PROGRAM P_U01
VAR_INPUT
	auto_mode_on														: BOOL;

	shutdown_process													: BOOL;
	{attribute 'OPC.UA.DA' := '1'}  				                
	{attribute 'OPC.UA.DA.Access' := '1'}  				                
	co2_adsorption_interlock											: BOOL;
    /// <summary>PCV01</summary>
	{attribute 'OPC.UA.DA' := '1'}  				                
	vacuum_pres_control_valve											: REAL;
    /// <summary>PCV01</summary>                  	           
	{attribute 'OPC.UA.DA' := '1'}  				                
	vacuum_pres_control_valve_mode										: INT;			
    /// <summary>PCV02</summary>
	{attribute 'OPC.UA.DA' := '1'}  				                
	steam_flow_control_valve											: REAL;
    /// <summary>PCV02</summary>                  	           
	{attribute 'OPC.UA.DA' := '1'}  				                
	steam_flow_control_valve_mode										: INT;			
	{attribute 'OPC.UA.DA' := '1'}  				                
	{attribute 'OPC.UA.DA.Access' := '1'}  				                
	hot_sorbent_for_repressurization_interlock							: BOOL;
	{attribute 'OPC.UA.DA' := '1'}  				                
	{attribute 'OPC.UA.DA.Access' := '1'}  				                
	drainage_on															: BOOL;
	{attribute 'OPC.UA.DA' := '1'}  				                
	{attribute 'OPC.UA.DA.Access' := '1'}  				                
	repressurization_valve_with_steam_interlock							: BOOL;
	{attribute 'OPC.UA.DA' := '1'}  				                
	{attribute 'OPC.UA.DA.Access' := '1'}  				                
	door_open_with_steam_flow_interlock									: BOOL;
	{attribute 'OPC.UA.DA' := '1'}  				                
	{attribute 'OPC.UA.DA.Access' := '1'}  				                
	door_open_with_reactor_vacuum_interlock								: BOOL;
	{attribute 'OPC.UA.DA' := '1'}  				                
	{attribute 'OPC.UA.DA.Access' := '1'}  				                
	hot_reactor_condenser_interlock										: BOOL;
	{attribute 'OPC.UA.DA' := '1'}  				                
	{attribute 'OPC.UA.DA.Access' := '1'}  				                
	no_steam_unevacuated_reactor_interlock								: BOOL;
	{attribute 'OPC.UA.DA' := '1'}  				                
	{attribute 'OPC.UA.DA.Access' := '1'}  				                
	reactor_over_safe_pressure_limit_interlock							: BOOL;
	{attribute 'OPC.UA.DA' := '1'}  				                
	{attribute 'OPC.UA.DA.Access' := '1'}  				                
	reactor_over_safe_temperature_limit_interlock						: BOOL;
	
	/// <summary>XV10</summary>
	{attribute 'OPC.UA.DA' := '1'}  				                
	dead_air_inlet_valve												: BOOL;
	/// <summary>XV11</summary>
	{attribute 'OPC.UA.DA' := '1'}  				                
	product_line_ambient_valve											: BOOL;
    /// <summary>X01</summary>
	{attribute 'OPC.UA.DA' := '1'}  				                
	vacuum_liquid_loop_fan												: BOOL;
    /// <summary>P05</summary>
	{attribute 'OPC.UA.DA' := '1'}  				                
	vacuum_liquid_pump													: BOOL;
    /// <summary>P02</summary>
	{attribute 'OPC.UA.DA' := '1'}  				                
	vacuum_pump															: BOOL;
    /// <summary>XV04</summary>
	{attribute 'OPC.UA.DA' := '1'}  				                
	vacuum_pump_bypass_valve											: BOOL;
    /// <summary>XV03</summary>
	{attribute 'OPC.UA.DA' := '1'}  				                
	vacuum_pump_inlet_valve												: BOOL;
    /// <summary>P01</summary>
	{attribute 'OPC.UA.DA' := '1'}  				                
	steam_water_pump													: BOOL;
    /// <summary>B01</summary>
	{attribute 'OPC.UA.DA' := '1'}  				                
	boiler_package														: BOOL;
    /// <summary>P04</summary>
	{attribute 'OPC.UA.DA' := '1'}  				                
	condenser_pump														: BOOL;
    /// <summary>E01</summary>
	{attribute 'OPC.UA.DA' := '1'}  				                
	condenser_fan														: BOOL;
    /// <summary>P06</summary>
	{attribute 'OPC.UA.DA' := '1'}  				                
	vacuum_separator_drain_pump											: BOOL;
    /// <summary>PCV02</summary>
	steam_flow_control_valve_setpoint									: REAL;
	condenser_knockout_drain_adsorption_on									: BOOL;
	
END_VAR
VAR_OUTPUT
	utility_error														: STRING;
    /// <summary>XV10</summary>
	dead_air_inlet_valve_clear											: BOOL;
    /// <summary>XV11</summary>
	product_line_ambient_valve_clear									: BOOL;
    /// <summary>XV03</summary>
	vacuum_pump_inlet_valve_clear										: BOOL;
END_VAR
VAR

	fbWriteData															: FB_WritePersistentData;
	tonWriteData														: TON;
	bWriteData															: BOOL;
	
	sError																: STRING;
	sMessage															: STRING;
	sUtilityError														: STRING;
	sRS																	: STRING;
	iAxStep																: INT;
	i2Step																: INT;
	i3Step																: INT;
	i8Step																: INT;
	i9Step																: INT;
	iVfd_Speed															: INT;
	bCondition1															: BOOL;
	bCondition2															: BOOL;
	bCondition3															: BOOL;
	bAdsorptionActive													: BOOL;
	bComplete															: BOOL;
	bPreCheckDone														: BOOL;
	bTimer																: BOOL;
	bPass1																: BOOL;
	bPass2																: BOOL;
	bPass3																: BOOL;
	bAdsorptionTimer													: BOOL;
	bCloseXVValves														: BOOL;
	bRunSteamBypass														: BOOL;
	bVfd_Speed_Up														: BOOL;
	bCondenserKnockoutError												: BOOL;
	bVacuumSeparatorFillError											: BOOL;
	bVacuumSeparatorDrainError											: BOOL;
	rTime																: REAL;
	rSP																	: REAL;
	rPres																: REAL;
	tonTimer															: TON;
	tonAdsorptionTimer													: TON;
	tonBoilerCheck														: TON;
	tonVacuumInterlock													: TON;
	tonCondenserKODrain													: TON;
	tonVacuumSeparatorFill												: TON;
	tonVacuumSeparatorDrain												: TON;
	rtrigVacuumSeparator												: R_TRIG;
	rtrigKODrainValve													: R_TRIG;
	
	bCondenserFlowError													: BOOL;
	bCondensateFlowError												: BOOL;
	bFlowCalibrationDiffPresError										: BOOL;
	bInletLineTempError                                  	            : BOOL;
	bProductOutletCo2Error												: BOOL;
	bProductOutletFlowError												: BOOL;
	bProductOutletH2oError												: BOOL;
	bProductTempError                                   		       	: BOOL;
	bProductVacuumPresError												: BOOL;
	bProductVacuumTempError                              	          	: BOOL;
	bSteamFlowError														: BOOL;
	bSteamLinePresError													: BOOL;
	bSteamWaterTankLevelError											: BOOL;
	bVacuumPumpWaterFlowError											: BOOL;
	bVacuumPumpWaterTemp1Error											: BOOL;
	bVacuumSeparatorLevelError											: BOOL;
	bWaterFeedFlowError													: BOOL;
	bWaterScale1Error													: BOOL;
	bWaterScale2Error													: BOOL;
	bWaterScale3Error													: BOOL;

	fb_Vacuum_Pres_Control_Valve_PI										: FB_PI_Control();
	fb_Steam_Flow_Control_Valve_PI										: FB_PI_Control();
	
	fb_WaterScales_In													: FB_RateOfChange;
 	fb_WaterScales_Out													: FB_RateOfChange;
	{attribute 'OPC.UA.DA' := '1'} 
	water_scales_in_delta												: REAL;
	{attribute 'OPC.UA.DA' := '1'} 
	water_scales_out_delta												: REAL;
	{attribute 'OPC.UA.DA' := '1'} 
	water_scales_in_rate												: REAL;
	{attribute 'OPC.UA.DA' := '1'} 
	water_scales_out_rate												: REAL;
	{attribute 'OPC.UA.DA' := '1'} 
	water_scales_reset													: BOOL;
	fb_adsorp_product_wastewater										: FB_ChangeOfValue;
	
	{attribute 'OPC.UA.DA' := '1'}  				                
	pressure_drop_test													: BOOL;							// Pressure drop test flag

	{attribute 'OPC.UA.DA' := '1'}  				                
	interlock_condenser_steam_or										: BOOL;							// Override condenser pump & fan needing to be on when steam is flowing
	{attribute 'OPC.UA.DA' := '1'}  				                
	{attribute 'OPC.UA.DA.Access' := '1'}  				                
	interlock_condenser_steam_or_status									: BOOL;
	{attribute 'OPC.UA.DA' := '1'}  				                
	{attribute 'OPC.UA.DA.Access' := '1'}  				                
	condenser_steam_interlock											: BOOL;
	
	{attribute 'OPC.UA.DA' := '1'}  				                
	interlock_hot_reactor_condenser_or									: BOOL;							// Override dead air valve needing to be open if sorbent temp is high
	{attribute 'OPC.UA.DA' := '1'}  				                
	{attribute 'OPC.UA.DA.Access' := '1'}  				                
	interlock_hot_reactor_condenser_or_status							: BOOL;
	
	{attribute 'OPC.UA.DA' := '1'}  				                
	interlock_no_steam_unevacuated_reactor_or							: BOOL;							// Override no steam to unevacuated reactor
	{attribute 'OPC.UA.DA' := '1'}  				                
	{attribute 'OPC.UA.DA.Access' := '1'}  				                
	interlock_no_steam_unevacuated_reactor_or_status					: BOOL;
	
	{attribute 'OPC.UA.DA' := '1'}  				                
	interlock_cooling_with_vacuum_or									: BOOL;							// Override vacuum not running without cooling loop active
	{attribute 'OPC.UA.DA' := '1'}  				                
	{attribute 'OPC.UA.DA.Access' := '1'}  				                
	interlock_cooling_with_vacuum_or_status								: BOOL;
	{attribute 'OPC.UA.DA' := '1'}  				                
	{attribute 'OPC.UA.DA.Access' := '1'}  				                
	cooling_with_vacuum_interlock										: BOOL;
	
	{attribute 'OPC.UA.DA' := '1'}  				                
	interlock_separator_water_level_with_vacuum_or						: BOOL;							// Override vacuum not running while separator water level too high or too low
	{attribute 'OPC.UA.DA' := '1'}  				                
	{attribute 'OPC.UA.DA.Access' := '1'}  				                
	interlock_separator_water_level_with_vacuum_or_status				: BOOL;
	{attribute 'OPC.UA.DA' := '1'}  				                
	{attribute 'OPC.UA.DA.Access' := '1'}  				                
	separator_water_level_with_vacuum_interlock							: BOOL;
	
	{attribute 'OPC.UA.DA' := '1'}  				                
	interlock_cooling_loop_flow_with_vacuum_or							: BOOL;							// Override vacuum not running with insufficient cooling flow
	{attribute 'OPC.UA.DA' := '1'}  				                
	{attribute 'OPC.UA.DA.Access' := '1'}  				                
	interlock_cooling_loop_flow_with_vacuum_or_status					: BOOL;
	{attribute 'OPC.UA.DA' := '1'}  				                
	{attribute 'OPC.UA.DA.Access' := '1'}  				                
	cooling_loop_flow_with_vacuum_interlock								: BOOL;
	
	{attribute 'OPC.UA.DA' := '1'}  				                
	interlock_condensate_tank_level_for_steam_or						: BOOL;							// Override steam not running with condensate collection tank low 
	{attribute 'OPC.UA.DA' := '1'}  				                
	{attribute 'OPC.UA.DA.Access' := '1'}  				                
	interlock_condensate_tank_level_for_steam_or_status					: BOOL;
	{attribute 'OPC.UA.DA' := '1'}  				                
	{attribute 'OPC.UA.DA.Access' := '1'}  				                
	condensate_tank_level_for_steam_interlock							: BOOL;
	
	{attribute 'OPC.UA.DA' := '1'}  				                
	interlock_hot_sorbent_for_repressurization_or						: BOOL;							// Override repressurization not running if sorbent temp is high 
	{attribute 'OPC.UA.DA' := '1'}  				                
	{attribute 'OPC.UA.DA.Access' := '1'}  				                
	interlock_hot_sorbent_for_repressurization_or_status				: BOOL;
	
	{attribute 'OPC.UA.DA' := '1'}  				                
	interlock_reactor_over_safe_pressure_limit_or						: BOOL;							// Override reactor over safe pressure limit
	{attribute 'OPC.UA.DA' := '1'}  				                
	{attribute 'OPC.UA.DA.Access' := '1'}  				                
	interlock_reactor_over_safe_pressure_limit_or_status				: BOOL;
	
	{attribute 'OPC.UA.DA' := '1'}  				                
	interlock_reactor_over_safe_temperature_limit_or					: BOOL;							// Override reactor over safe temperature limit
	{attribute 'OPC.UA.DA' := '1'}  				                
	{attribute 'OPC.UA.DA.Access' := '1'}  				                
	interlock_reactor_over_safe_temperature_limit_or_status				: BOOL;
	
	{attribute 'OPC.UA.DA' := '1'}  				                
	interlock_repressurization_valve_with_steam_or						: BOOL;							// Override repressurization valve with steam flow
	{attribute 'OPC.UA.DA' := '1'}  				                
	{attribute 'OPC.UA.DA.Access' := '1'}  				                
	interlock_repressurization_valve_with_steam_or_status				: BOOL;
	
	{attribute 'OPC.UA.DA' := '1'}  				                
	interlock_door_open_with_steam_flow_or								: BOOL;							// Override door open with steam flow
	{attribute 'OPC.UA.DA' := '1'}  				                
	{attribute 'OPC.UA.DA.Access' := '1'}  				                
	interlock_door_open_with_steam_flow_or_status						: BOOL;
	
	{attribute 'OPC.UA.DA' := '1'}  				                
	interlock_door_open_with_reactor_vacuum_or							: BOOL;							// Override door open with reactor under vacuum
	{attribute 'OPC.UA.DA' := '1'}  				                
	{attribute 'OPC.UA.DA.Access' := '1'}  				                
	interlock_door_open_with_reactor_vacuum_or_status					: BOOL;
	
	{attribute 'OPC.UA.DA' := '1'}  				                
	interlock_co2_adsorption_or											: BOOL;							// Override co2 adsorption solenoids
	{attribute 'OPC.UA.DA' := '1'}  				                
	{attribute 'OPC.UA.DA.Access' := '1'}  				                
	interlock_co2_adsorption_or_status									: BOOL;
	
	{attribute 'OPC.UA.DA' := '1'}  				                
	interlock_condensate_pump_or										: BOOL;							// Override condensate pump
	{attribute 'OPC.UA.DA' := '1'}  				                
	{attribute 'OPC.UA.DA.Access' := '1'}  				                
	interlock_condensate_pump_or_status									: BOOL;
	{attribute 'OPC.UA.DA' := '1'}  				                
	{attribute 'OPC.UA.DA.Access' := '1'}  				                
	interlock_condensate_pump											: BOOL;
	
	{attribute 'OPC.UA.DA' := '1'}  				                
	vacuum_separator_drain_or_on										: BOOL;
	{attribute 'OPC.UA.DA' := '1'}  				                
	{attribute 'OPC.UA.DA.Access' := '1'}  				                
	vacuum_separator_drain_or_on_status									: BOOL;
	{attribute 'OPC.UA.DA' := '1'}  				                
	vacuum_separator_drain_or_off										: BOOL;
	{attribute 'OPC.UA.DA' := '1'}  				                
	{attribute 'OPC.UA.DA.Access' := '1'}  				                
	vacuum_separator_drain_or_off_status								: BOOL;

	{attribute 'OPC.UA.DA' := '1'}  				                
	reactor_drain_or_on													: BOOL;
	{attribute 'OPC.UA.DA' := '1'}  				                
	{attribute 'OPC.UA.DA.Access' := '1'}  				                
	reactor_drain_or_on_status											: BOOL;
	{attribute 'OPC.UA.DA' := '1'}  				                
	reactor_drain_or_off												: BOOL;
	{attribute 'OPC.UA.DA' := '1'}  				                
	{attribute 'OPC.UA.DA.Access' := '1'}  				                
	reactor_drain_or_off_status											: BOOL;

	{attribute 'OPC.UA.DA' := '1'}  				                
	condenser_knockout_drain_or_on										: BOOL;
	{attribute 'OPC.UA.DA' := '1'}  				                
	{attribute 'OPC.UA.DA.Access' := '1'}  				                
	condenser_knockout_drain_or_on_status								: BOOL;
	{attribute 'OPC.UA.DA' := '1'}  				                
	condenser_knockout_drain_or_off										: BOOL;
	{attribute 'OPC.UA.DA' := '1'}  				                
	{attribute 'OPC.UA.DA.Access' := '1'}  				                
	condenser_knockout_drain_or_off_status								: BOOL;

	{attribute 'OPC.UA.DA' := '1'}  				                
	{attribute 'OPC.UA.DA.Access' := '1'}  				                
	warmup_complete														: BOOL;
	{attribute 'OPC.UA.DA' := '1'}  				                
	{attribute 'OPC.UA.DA.Access' := '1'}  				                
	steam_bypass_complete												: BOOL;

	{attribute 'OPC.UA.DA' := '1'}  				                
	write_persistent_data												: BOOL;
	{attribute 'OPC.UA.DA' := '1'}  				                
	drainage_function_on_or												: BOOL;
	{attribute 'OPC.UA.DA' := '1'}  				                
	drainage_function_off_or											: BOOL;
	
	
	// PIDs
	steam_valve_pid 												: FB_CTRL_PID;
	steam_valve_pid_params											: ST_CTRL_PID_PARAMS;
	steam_valve_pid_mode											: E_CTRL_MODE := E_CTRL_MODE.eCTRL_MODE_MANUAL;
	steam_valve_pid_manual_sp										: LREAL := 50;   // Pressure SP value in manual mode
	steam_valve_pid_sp_value										: LREAL;  // Pressure SP value
	steam_valve_pid_actual_value									: LREAL;  // Presure Actual Value
	steam_valve_pid_out												: LREAL;  // valve control signal ( 0-100 %)
	steam_valve_pid_simulate_timer									: TON;
	steam_valve_pid_kp												: LREAL := 0.5;
	steam_valve_pid_tn												: TIME := T#5S;
	steam_valve_pid_tv												: TIME := T#0S;
	
	
	simulate_process												: FB_CTRL_PT2oscillation;
	simulate_process_params											: ST_CTRL_PT2oscillation_PARAMS ;
	simulate_process_kp												: REAL := 20;
	simulate_process_dumping_ration									: REAL := 0.5;
	simulate_process_tT0											: REAL := 0;
	
//	fb_MovingAverage												: FB_CTRL_MOVING_AVERAGE;
	moving_avg_in													: REAL;
	moving_avg_out													: LREAL;
	moving_avg_params												: ST_CTRL_MOVING_AVERAGE_PARAMS;
	moving_avg_array												: ARRAY[1..10] OF REAL;
	moving_avg_in_sim_timer											: TON;
	
	fbMovingAverage													: FB_MovingAverage;
	
	condenser_tank_capacity										: REAL;
	steam_delivery_tank_capacity										: REAL;
	condenser_tank_room_before_full										: REAL;
	steam_delivery_tank_before_empty										: REAL;
	
    /// <summary>LS01</summary>
	{attribute 'OPC.UA.DA' := '1'}  				                
	{attribute 'OPC.UA.DA.Access' := '1'}  				                
	product_condensate_drum_lsl									AT %I*	: BOOL;
    /// <summary>LS02</summary>
	{attribute 'OPC.UA.DA' := '1'}  				                
	{attribute 'OPC.UA.DA.Access' := '1'}  				                
	product_condensate_drum_lsh									AT %I*	: BOOL;

    /// <summary>B01</summary>
	{attribute 'OPC.UA.DA' := '1'}  				                
	{attribute 'OPC.UA.DA.Access' := '1'}  				                
	boiler_package_cmd_status											: BOOL;
    /// <summary>B01</summary>
	{attribute 'OPC.UA.DA' := '1'}  				                
	boiler_ready														: BOOL;
    /// <summary>boiler package</summary>
	B_01														AT %Q*	: BOOL;
    /// <summary>B01</summary>
	{attribute 'OPC.UA.DA' := '1'}  				                
	boiler_reset												AT %Q*	: BOOL;
	
    /// <summary>P02</summary>
	{attribute 'OPC.UA.DA' := '1'}  				                
	{attribute 'OPC.UA.DA.Access' := '1'}  				                
	steam_water_pump_cmd_status											: BOOL;
    /// <summary>vacuum pump</summary>
	P_01														AT %Q*	: BOOL;

    /// <summary>P02</summary>
	{attribute 'OPC.UA.DA' := '1'}  				                
	{attribute 'OPC.UA.DA.Access' := '1'}  				                
	vacuum_pump_cmd_status												: BOOL;
    /// <summary>vacuum pump</summary>
	P_02														AT %Q*	: BOOL;

    /// <summary>P03</summary>
	{attribute 'OPC.UA.DA' := '1'}  				                
	condensate_pump														: BOOL;
    /// <summary>P03</summary>
	{attribute 'OPC.UA.DA' := '1'}  				                
	{attribute 'OPC.UA.DA.Access' := '1'}  				                
	condensate_pump_cmd_status											: BOOL;
    /// <summary>condensate pump</summary>
	P_03														AT %Q*	: BOOL;

    /// <summary>P04</summary>
	{attribute 'OPC.UA.DA' := '1'}  				                
	{attribute 'OPC.UA.DA.Access' := '1'}  				                
	condenser_pump_cmd_status											: BOOL;
    /// <summary>condenser pump</summary>
	P_04														AT %Q*	: BOOL;

    /// <summary>P05</summary>
	{attribute 'OPC.UA.DA' := '1'}  				                
	{attribute 'OPC.UA.DA.Access' := '1'}  				                
	vacuum_liquid_pump_cmd_status										: BOOL;
    /// <summary>vacuum liquid pump</summary>
	P_05														AT %Q*	: BOOL;

    /// <summary>P06</summary>
	{attribute 'OPC.UA.DA' := '1'}  				                
	{attribute 'OPC.UA.DA.Access' := '1'}  				                
	vacuum_separator_drain_pump_cmd_status								: BOOL;
    /// <summary>vacuum cooling pump</summary>
	P_06														AT %Q*	: BOOL;

    /// <summary>E01</summary>
	{attribute 'OPC.UA.DA' := '1'}  				                
	{attribute 'OPC.UA.DA.Access' := '1'}  				                
	condenser_fan_cmd_status											: BOOL;
    /// <summary>condenser fan</summary>
	E_01														AT %Q*	: BOOL;

    /// <summary>X01</summary>
	{attribute 'OPC.UA.DA' := '1'}  				                
	{attribute 'OPC.UA.DA.Access' := '1'}  				                
	vacuum_liquid_loop_fan_cmd_status									: BOOL;
    /// <summary>vacuum liquid loop fan</summary>
	X_01														AT %Q*	: BOOL;

    /// <summary>AT02</summary>
	{attribute 'OPC.UA.DA' := '1'}  				                
	{attribute 'OPC.UA.DA.Access' := '1'}  				                
	product_outlet_co2													: REAL;
	{attribute 'OPC.UA.DA' := '1'}  				                
	{attribute 'OPC.UA.DA.Access' := '1'} 
    /// <summary>AT02</summary>
	product_outlet_co2_error											: BOOL;
    /// <summary>product outlet co2</summary>
	{attribute 'OPC.UA.DA' := '1'}  				                
	_ProductOutletCO2ErrorOff											: BOOL;
    /// <summary>AT02</summary>
	{attribute 'OPC.UA.DA' := '1'}  				                
	AT_02														AT %I*	: INT;
    /// <summary>AT02</summary>
	{attribute 'OPC.UA.DA' := '1'}  				                
	{attribute 'OPC.UA.DA.Access' := '1'}  				                
	AT_02_error													AT %I*	: BOOL;
    
	/// <summary>AT03</summary>
	{attribute 'OPC.UA.DA' := '1'}  				                
	{attribute 'OPC.UA.DA.Access' := '1'}  				                
	product_outlet_h2o													: REAL;
    /// <summary>AT03</summary>
	{attribute 'OPC.UA.DA' := '1'}  				                
	{attribute 'OPC.UA.DA.Access' := '1'}  				                
	product_outlet_h2o_error											: BOOL;
	/// <summary>AT03</summary>
	{attribute 'OPC.UA.DA' := '1'}  				                
	_ProductOutletH2OErrorOff											: BOOL;
    /// <summary>product outlet h2o</summary>
	AT_03														AT %I*	: INT;
    /// <summary>product outlet h2o</summary>
	{attribute 'OPC.UA.DA' := '1'}  				                
	{attribute 'OPC.UA.DA.Access' := '1'}  				                
	AT_03_error													AT %I*	: BOOL;

    /// <summary>FT02</summary>
	{attribute 'OPC.UA.DA' := '1'}  				                
	{attribute 'OPC.UA.DA.Access' := '1'}  					                
	product_outlet_flow													: REAL;
    /// <summary>FT02</summary>
	{attribute 'OPC.UA.DA' := '1'}  				                
	{attribute 'OPC.UA.DA.Access' := '1'}  				                
	product_outlet_flow_error											: BOOL;
    /// <summary>FT02</summary>
	{attribute 'OPC.UA.DA' := '1'}  				                
	_ProductOutletFlowErrorOff											: BOOL;
    /// <summary>product outlet flow</summary>
	FT_02														AT %I*	: INT;
    /// <summary>product outlet flow</summary>
	{attribute 'OPC.UA.DA' := '1'}  				                
	{attribute 'OPC.UA.DA.Access' := '1'}  				                
	FT_02_error													AT %I*	: BOOL;

    /// <summary>FT04</summary>
	{attribute 'OPC.UA.DA' := '1'}  				                
	{attribute 'OPC.UA.DA.Access' := '1'}  				                
	condensate_flow														: REAL;
    /// <summary>FT04</summary>
	{attribute 'OPC.UA.DA' := '1'}  				                
	{attribute 'OPC.UA.DA.Access' := '1'}  				                
	condensate_flow_error												: BOOL;
    /// <summary>FT04</summary>
	{attribute 'OPC.UA.DA' := '1'}  				                
	_CondensateFlowErrorOff												: BOOL;
    /// <summary>condensate flow</summary>
	FT_04														AT %I*	: INT;
    /// <summary>condensate flow</summary>
	{attribute 'OPC.UA.DA' := '1'}  				                
	{attribute 'OPC.UA.DA.Access' := '1'}  				                
	FT_04_error													AT %I*	: BOOL;

    /// <summary>FT05</summary>
	{attribute 'OPC.UA.DA' := '1'}  				                
	{attribute 'OPC.UA.DA.Access' := '1'}  					                
	tap_water_feed_flow													: REAL;
    /// <summary>FT05</summary>
	{attribute 'OPC.UA.DA' := '1'}  				                
	{attribute 'OPC.UA.DA.Access' := '1'}  				                
	tap_water_feed_flow_error											: BOOL;
    /// <summary>FT05</summary>
	{attribute 'OPC.UA.DA' := '1'}  				                
	_TapWaterFeedFlowErrorOff											: BOOL;
    /// <summary>tap water feed flow</summary>
	FT_05														AT %I*	: INT;
    /// <summary>tap water feed flow</summary>
	{attribute 'OPC.UA.DA' := '1'}  				                
	{attribute 'OPC.UA.DA.Access' := '1'}  				                
	FT_05_error													AT %I*	: BOOL;

    /// <summary>FT06</summary>
	{attribute 'OPC.UA.DA' := '1'}  				                
	{attribute 'OPC.UA.DA.Access' := '1'}  					                
	steam_flow															: REAL;
    /// <summary>FT06</summary>
	{attribute 'OPC.UA.DA' := '1'}  				                
	{attribute 'OPC.UA.DA.Access' := '1'}  				                
	steam_flow_error													: BOOL;
    /// <summary>FT06</summary>
	{attribute 'OPC.UA.DA' := '1'}  				                
	_SteamFlowErrorOff													: BOOL;
    /// <summary>steam flow</summary>
	FT_06														AT %I*	: INT;
    /// <summary>steam flow</summary>
	{attribute 'OPC.UA.DA' := '1'}  				                
	{attribute 'OPC.UA.DA.Access' := '1'}  				                
	FT_06_error													AT %I*	: BOOL;

    /// <summary>FT07</summary>
	{attribute 'OPC.UA.DA' := '1'}  				                
	{attribute 'OPC.UA.DA.Access' := '1'}  					                
	vacuum_pump_water_flow												: REAL;
    /// <summary>FT07</summary>
	{attribute 'OPC.UA.DA' := '1'}  				                
	{attribute 'OPC.UA.DA.Access' := '1'}  				                
	vacuum_pump_water_flow_error										: BOOL;
    /// <summary>FT07</summary>
	{attribute 'OPC.UA.DA' := '1'}  				                
	_VacuumPumpWaterFlowErrorOff										: BOOL;
    /// <summary>vacuum pump water flow</summary>
	FT_07														AT %I*	: INT;
    /// <summary>vacuum pump water flow</summary>
    /// <summary>FT07</summary>
	{attribute 'OPC.UA.DA' := '1'}  				                
	{attribute 'OPC.UA.DA.Access' := '1'}  				                
	FT_07_error													AT %I*	: BOOL;

    /// <summary>FT08</summary>
	{attribute 'OPC.UA.DA' := '1'}  				                
	{attribute 'OPC.UA.DA.Access' := '1'}  					                
	condenser_flow														: REAL;
    /// <summary>FT08</summary>
	{attribute 'OPC.UA.DA' := '1'}  				                
	{attribute 'OPC.UA.DA.Access' := '1'}  				                
	condenser_flow_error												: BOOL;
    /// <summary>FT08</summary>
	{attribute 'OPC.UA.DA' := '1'}  				                
	_CondenserFlowErrorOff												: BOOL;
    /// <summary>vacuum pump water flow</summary>
	FT_08														AT %I*	: INT;
    /// <summary>vacuum pump water flow</summary>
    /// <summary>FT08</summary>
	{attribute 'OPC.UA.DA' := '1'}  				                
	{attribute 'OPC.UA.DA.Access' := '1'}  				                
	FT_08_error													AT %I*	: BOOL;

    /// <summary>LT01</summary>
	{attribute 'OPC.UA.DA' := '1'}  				                
	{attribute 'OPC.UA.DA.Access' := '1'}  					                
	steam_water_tank_level												: REAL;
    /// <summary>LT01</summary>
	{attribute 'OPC.UA.DA' := '1'}  				                
	{attribute 'OPC.UA.DA.Access' := '1'}  				                
	steam_water_tank_level_error										: BOOL;
    /// <summary>LT01</summary>
	{attribute 'OPC.UA.DA' := '1'}  				                
	_SteamWaterTankLevelErrorOff										: BOOL;
    /// <summary>steam water tank level</summary>
	LT_01														AT %I*	: INT;
    /// <summary>steam water tank level</summary>
    /// <summary>LT01</summary>
	{attribute 'OPC.UA.DA' := '1'}  				                
	{attribute 'OPC.UA.DA.Access' := '1'}  				                
	LT_01_error													AT %I*	: BOOL;

    /// <summary>LT02</summary>
	{attribute 'OPC.UA.DA' := '1'}  				                
	{attribute 'OPC.UA.DA.Access' := '1'}  					                
	vacuum_separator_level												: REAL;
    /// <summary>LT02</summary>
	{attribute 'OPC.UA.DA' := '1'}  				                
	{attribute 'OPC.UA.DA.Access' := '1'}  				                
	vacuum_separator_level_error										: BOOL;
    /// <summary>LT02</summary>
	{attribute 'OPC.UA.DA' := '1'}  				                
	_VacuumSeparatorLevelErrorOff										: BOOL;
    /// <summary>vacuum separator level</summary>
	LT_02														AT %I*	: INT;
    /// <summary>vacuum separator level</summary>
    /// <summary>LT02</summary>
	{attribute 'OPC.UA.DA' := '1'}  				                
	{attribute 'OPC.UA.DA.Access' := '1'}  				                
	LT_02_error													AT %I*	: BOOL;

    /// <summary>PT04</summary>
	{attribute 'OPC.UA.DA' := '1'}  				                
	{attribute 'OPC.UA.DA.Access' := '1'}  				                
	product_vacuum_pres													: REAL;
    /// <summary>PT04</summary>
	{attribute 'OPC.UA.DA' := '1'}  				                
	{attribute 'OPC.UA.DA.Access' := '1'}  				                
	product_vacuum_pres_error											: BOOL;
    /// <summary>PT04</summary>
	{attribute 'OPC.UA.DA' := '1'}  				                
	_ProductVacuumPresErrorOff											: BOOL;
    /// <summary>product vacuum pres</summary>
	PT_04														AT %I*	: INT;
    /// <summary>product vacuum pres</summary>
    /// <summary>PT04</summary>
	{attribute 'OPC.UA.DA' := '1'}  				                
	{attribute 'OPC.UA.DA.Access' := '1'}  				                
	PT_04_error													AT %I*	: BOOL;

    /// <summary>PT07</summary>
	{attribute 'OPC.UA.DA' := '1'}  				                
	{attribute 'OPC.UA.DA.Access' := '1'}  				                
	steam_line_pres														: REAL;
    /// <summary>PT07</summary>
	{attribute 'OPC.UA.DA' := '1'}  				                
	{attribute 'OPC.UA.DA.Access' := '1'}  				                
	steam_line_pres_error												: BOOL;
    /// <summary>PT07</summary>
	{attribute 'OPC.UA.DA' := '1'}  				                
	_SteamLinePresErrorOff												: BOOL;
    /// <summary>steam line pres</summary>
	PT_07														AT %I*	: INT;
    /// <summary>steam line pres</summary>
	{attribute 'OPC.UA.DA' := '1'}  				                
	{attribute 'OPC.UA.DA.Access' := '1'}  				                
	PT_07_error													AT %I*	: BOOL;

    /// <summary>PDT04</summary>
	{attribute 'OPC.UA.DA' := '1'}  				                
	{attribute 'OPC.UA.DA.Access' := '1'}  				                
	flow_calibration_diff_pres											: REAL;
    /// <summary>PDT04</summary>
	{attribute 'OPC.UA.DA' := '1'}  				                
	{attribute 'OPC.UA.DA.Access' := '1'}  				                
	flow_calibration_diff_pres_error									: BOOL;
    /// <summary>PDT04</summary>
	{attribute 'OPC.UA.DA' := '1'}  				                
	_FlowCalibrationDiffPresErrorOff									: BOOL;
    /// <summary>flow calibration diff pres</summary>
	PDT_04														AT %I*	: INT;
    /// <summary>flow calibration diff pres</summary>
	{attribute 'OPC.UA.DA' := '1'}  				                
	{attribute 'OPC.UA.DA.Access' := '1'}  				                
	PDT_04_error												AT %I*	: BOOL;

    /// <summary>TT02</summary>
	{attribute 'OPC.UA.DA' := '1'}  				                
	{attribute 'OPC.UA.DA.Access' := '1'}  				                
	product_temp														: REAL;
    /// <summary>TT02</summary>
	{attribute 'OPC.UA.DA' := '1'}  				                
	{attribute 'OPC.UA.DA.Access' := '1'}  				                
	product_temp_error													: BOOL;
	{attribute 'OPC.UA.DA' := '1'}  				                
	_ProductTempErrorOff												: BOOL;
    /// <summary>product temp</summary>
	TT_02														AT %I*	: INT;
    /// <summary>product temp</summary>
	{attribute 'OPC.UA.DA' := '1'}  				                
	{attribute 'OPC.UA.DA.Access' := '1'}  				                
	TT_02_error													AT %I*	: BOOL;

    /// <summary>TT03</summary>
	{attribute 'OPC.UA.DA' := '1'}  				                
	{attribute 'OPC.UA.DA.Access' := '1'}  				                
	product_vacuum_temp													: REAL;
    /// <summary>TT03</summary>
	{attribute 'OPC.UA.DA' := '1'}  				                
	{attribute 'OPC.UA.DA.Access' := '1'}  				                
	product_vacuum_temp_error											: BOOL;
    /// <summary>TT03</summary>
	{attribute 'OPC.UA.DA' := '1'}  				                
	_ProductVacuumTempOff												: BOOL;
    /// <summary>product vacuum temp</summary>
	TT_03														AT %I*	: INT;
    /// <summary>product vacuum temp</summary>
	{attribute 'OPC.UA.DA' := '1'}  				                
	{attribute 'OPC.UA.DA.Access' := '1'}  				                
	TT_03_error													AT %I*	: BOOL;

    /// <summary>TT06</summary>
	{attribute 'OPC.UA.DA' := '1'}  				                
	{attribute 'OPC.UA.DA.Access' := '1'}  				                
	inlet_line_temp														: REAL;
    /// <summary>TT06</summary>
	{attribute 'OPC.UA.DA' := '1'}  				                
	{attribute 'OPC.UA.DA.Access' := '1'}  				                
	inlet_line_temp_error												: BOOL;
    /// <summary>TT06</summary>
	{attribute 'OPC.UA.DA' := '1'}  				                
	_InletLineTempErrorOff												: BOOL;
    /// <summary>inlet line temp</summary>
	TT_06														AT %I*	: INT;
    /// <summary>inlet line temp</summary>
	{attribute 'OPC.UA.DA' := '1'}  				                
	{attribute 'OPC.UA.DA.Access' := '1'}  				                
	TT_06_error													AT %I*	: BOOL;

    /// <summary>TT10</summary>
	{attribute 'OPC.UA.DA' := '1'}  				                
	{attribute 'OPC.UA.DA.Access' := '1'}  				                
	vacuum_pump_water_temp_1											: REAL;
    /// <summary>TT10</summary>
	{attribute 'OPC.UA.DA' := '1'}  				                
	{attribute 'OPC.UA.DA.Access' := '1'}  				                
	vacuum_pump_water_temp_1_error										: BOOL;
    /// <summary>TT10</summary>
	{attribute 'OPC.UA.DA' := '1'}  				                
	_VacuumPumpWaterTemp1ErrorOff										: BOOL;
    /// <summary>vacuum pump water temp 1</summary>
	TT_10														AT %I*	: INT;
    /// <summary>vacuum pump water temp 1</summary>
	{attribute 'OPC.UA.DA' := '1'}  				                
	{attribute 'OPC.UA.DA.Access' := '1'}  				                
	TT_10_error													AT %I*	: BOOL;
	
    /// <summary>TT11</summary>
	{attribute 'OPC.UA.DA' := '1'}  				                
	{attribute 'OPC.UA.DA.Access' := '1'}  				                
	vacuum_pump_water_temp_2											: REAL;
    /// <summary>TT11</summary>
	{attribute 'OPC.UA.DA' := '1'}  				                
	{attribute 'OPC.UA.DA.Access' := '1'}  				                
	vacuum_pump_water_temp_2_error										: BOOL;
    /// <summary>TT11</summary>
	{attribute 'OPC.UA.DA' := '1'}  				                
	_VacuumPumpWaterTemp2ErrorOff										: BOOL;
    /// <summary>vacuum pump water temp 2</summary>
	TT_11														AT %I*	: INT;
    /// <summary>vacuum pump water temp 2</summary>
	{attribute 'OPC.UA.DA' := '1'}  				                
	{attribute 'OPC.UA.DA.Access' := '1'}  				                
	TT_11_error													AT %I*	: BOOL;

    /// <summary>XV03</summary>
	{attribute 'OPC.UA.DA' := '1'}  				                
	{attribute 'OPC.UA.DA.Access' := '1'}  				                
	vacuum_pump_inlet_valve_open_cmd_status								: BOOL;
    /// <summary>XV03</summary>
	{attribute 'OPC.UA.DA' := '1'}  				                
	{attribute 'OPC.UA.DA.Access' := '1'}  				                
	vacuum_pump_inlet_valve_open								AT %I*	: BOOL;
    /// <summary>XV03</summary>
	{attribute 'OPC.UA.DA' := '1'}  				                
	{attribute 'OPC.UA.DA.Access' := '1'}  				                
	vacuum_pump_inlet_valve_closed								AT %I*	: BOOL;
    /// <summary>vacuum pump inlet valve</summary>
	XV_03														AT %Q*	: BOOL;
	
    /// <summary>XV04</summary>
	{attribute 'OPC.UA.DA' := '1'}  				                
	{attribute 'OPC.UA.DA.Access' := '1'}  				                
	vacuum_pump_bypass_valve_open_cmd_status							: BOOL;
    /// <summary>XV04</summary>
	{attribute 'OPC.UA.DA' := '1'}  				                
	{attribute 'OPC.UA.DA.Access' := '1'}  				                
	vacuum_pump_bypass_valve_open								AT %I*	: BOOL;
    /// <summary>XV04</summary>
	{attribute 'OPC.UA.DA' := '1'}  				                
	{attribute 'OPC.UA.DA.Access' := '1'}  				                
	vacuum_pump_bypass_valve_closed								AT %I*	: BOOL;
    /// <summary>vacuum pump bypass valve</summary>
	XV_04														AT %Q*	: BOOL;
    /// <summary>XV04</summary>
	vacuum_pump_bypass_valve_clear										: BOOL;
	
    /// <summary>XV06</summary>
	{attribute 'OPC.UA.DA' := '1'}  				                
	knockout_drain_valve												: BOOL;
    /// <summary>XV06</summary>
	{attribute 'OPC.UA.DA' := '1'}  				                
	{attribute 'OPC.UA.DA.Access' := '1'}  				                
	knockout_drain_valve_open_cmd_status								: BOOL;
    /// <summary>XV06</summary>
	{attribute 'OPC.UA.DA' := '1'}  				                
	{attribute 'OPC.UA.DA.Access' := '1'}  				                
	knockout_drain_valve_open									AT %I*	: BOOL;
    /// <summary>XV06</summary>
	{attribute 'OPC.UA.DA' := '1'}  				                
	{attribute 'OPC.UA.DA.Access' := '1'}  				                
	knockout_drain_valve_closed									AT %I*	: BOOL;
    /// <summary>knockout drain valve</summary>
	XV_06														AT %Q*	: BOOL;
    /// <summary>XV06</summary>
	knockout_drain_valve_clear											: BOOL;
	
    /// <summary>XV10</summary>
	{attribute 'OPC.UA.DA' := '1'}  				                
	{attribute 'OPC.UA.DA.Access' := '1'}  				                
	dead_air_inlet_valve_open_cmd_status								: BOOL;
    /// <summary>XV10</summary>
	{attribute 'OPC.UA.DA' := '1'}  				                
	{attribute 'OPC.UA.DA.Access' := '1'}  				                
	dead_air_inlet_valve_open									AT %I*	: BOOL;
    /// <summary>XV10</summary>
	{attribute 'OPC.UA.DA' := '1'}  				                
	{attribute 'OPC.UA.DA.Access' := '1'}  				                
	dead_air_inlet_valve_closed 								AT %I*	: BOOL;
    /// <summary>dead air inlet valve</summary>
	XV_10														AT %Q*	: BOOL;

    /// <summary>XV11</summary>
	{attribute 'OPC.UA.DA' := '1'}  				                
	{attribute 'OPC.UA.DA.Access' := '1'}  				                
	product_line_ambient_valve_cmd_status								: BOOL;
    /// <summary>XV11</summary>
	{attribute 'OPC.UA.DA' := '1'}  				                
	{attribute 'OPC.UA.DA.Access' := '1'}  				                
	product_line_ambient_valve_product 							AT %I*	: BOOL;				///@@@ Assuming open valve is Product
    /// <summary>XV11</summary>
	{attribute 'OPC.UA.DA' := '1'}  				                
	{attribute 'OPC.UA.DA.Access' := '1'}  				                
	product_line_ambient_valve_ambient							AT %I*	: BOOL;				///@@@ Assuming closed valve is Ambient
    /// <summary>product line ambient valve</summary>
	XV_11														AT %Q*	: BOOL;

	/// <summary>XV12</summary>
	{attribute 'OPC.UA.DA' := '1'}  				                
	tap_water_feed_valve												: BOOL;
    /// <summary>XV11</summary>
	{attribute 'OPC.UA.DA' := '1'}  				                
	{attribute 'OPC.UA.DA.Access' := '1'}  				                
	tap_water_feed_valve_cmd_status										: BOOL;
	XV_12														AT %Q*	: BOOL;

	/// <summary>XV13</summary>
	{attribute 'OPC.UA.DA' := '1'}  				                
	separator_drain_valve												: BOOL;
    /// <summary>XV13</summary>
	{attribute 'OPC.UA.DA' := '1'}  				                
	{attribute 'OPC.UA.DA.Access' := '1'}  				                
	separator_drain_valve_open_cmd_status								: BOOL;
    /// <summary>XV13</summary>
	{attribute 'OPC.UA.DA' := '1'}  				                
	{attribute 'OPC.UA.DA.Access' := '1'}  				                
	separator_drain_valve_open									AT %I*	: BOOL;
    /// <summary>XV13</summary>
	{attribute 'OPC.UA.DA' := '1'}  				                
	{attribute 'OPC.UA.DA.Access' := '1'}  				                
	separator_drain_valve_closed 								AT %I*	: BOOL;
    /// <summary>dead air inlet valve</summary>
	XV_13														AT %Q*	: BOOL;
    /// <summary>XV13</summary>
	separator_drain_valve_clear											: BOOL;

	/// <summary>XV14</summary>
	{attribute 'OPC.UA.DA' := '1'}  				                
	steam_water_reservoir_valve											: BOOL;
    /// <summary>XV14</summary>
	{attribute 'OPC.UA.DA' := '1'}  				                
	{attribute 'OPC.UA.DA.Access' := '1'}  				                
	steam_water_reservoir_valve_cmd_status								: BOOL;
    /// <summary>steam water reservoir valve</summary>
	XV_14														AT %Q*	: BOOL;

    /// <summary>PCV01</summary>
	vacuum_pres_control_valve_open										: BOOL;
    /// <summary>PCV01</summary>
	vacuum_pres_control_valve_closed									: BOOL;
    /// <summary>PCV01</summary>
	{attribute 'OPC.UA.DA' := '1'}  				                
	{attribute 'OPC.UA.DA.Access' := '1'}  				                
	vacuum_pres_control_valve_position									: REAL;
    /// <summary>PCV01</summary>
	{attribute 'OPC.UA.DA' := '1'}  				                
	{attribute 'OPC.UA.DA.Access' := '1'}  				                
	vacuum_pres_control_valve_position_error					AT %I*	: BOOL;
    /// <summary>vacuum pressure control valve</summary>
	PCV_01														AT %Q*	: INT;
    /// <summary>vacuum pressure control valve</summary>
	{attribute 'OPC.UA.DA' := '1'}  				                
	{attribute 'OPC.UA.DA.Access' := '1'}  				                
	PCV_01_position												AT %I*	: INT;
    /// <summary>PCV01</summary>                  	           
	{attribute 'OPC.UA.DA' := '1'}  				                
	{attribute 'OPC.UA.DA.Access' := '1'}  				                
	vacuum_pres_control_valve_current_mode								: INT;			
    /// <summary>PCV01</summary>                  	           
	vacuum_pres_control_valve_kp										: REAL		:= 0.01; 
    /// <summary>PCV01</summary>                  	           
	vacuum_pres_control_valve_ki										: REAL		:= 0.01;
    /// <summary>PCV01</summary>                  	           
	vacuum_pres_control_valve_loop_time									: REAL		:= 2000;
    /// <summary>PCV01</summary>                  	           
	vacuum_pres_control_valve_iband										: REAL		:= 6;
    /// <summary>PCV01</summary>                  	           
	vacuum_pres_control_valve_base										: INT		:= 13110;
    /// <summary>PCV01</summary>                  	           
	vacuum_pres_control_valve_base_adjust								: INT		:= 10;
	
    /// <summary>PCV02</summary>
	steam_flow_control_valve_open										: BOOL;
    /// <summary>PCV02</summary>
	steam_flow_control_valve_closed										: BOOL;
    /// <summary>PCV02</summary>
	{attribute 'OPC.UA.DA' := '1'}  				                
	{attribute 'OPC.UA.DA.Access' := '1'}  				                
	steam_flow_control_valve_position									: REAL;
    /// <summary>PCV02</summary>
	{attribute 'OPC.UA.DA' := '1'}  				                
	{attribute 'OPC.UA.DA.Access' := '1'}  				                
	steam_flow_control_valve_position_error								: BOOL;
    /// <summary>steam flow control valve</summary>
	PCV_02														AT %Q*	: INT;
    /// <summary>steam flow control valve</summary>
	{attribute 'OPC.UA.DA' := '1'}  				                
	{attribute 'OPC.UA.DA.Access' := '1'}  				                
	PCV_02_position												AT %I*	: INT;
    /// <summary>PCV02</summary>                  	           
	{attribute 'OPC.UA.DA' := '1'}  				                
	{attribute 'OPC.UA.DA.Access' := '1'}  				                
	steam_flow_control_valve_current_mode								: INT;			
    /// <summary>PCV02</summary>                  	           
	steam_flow_control_valve_kp											: REAL		:= 0.01; 
    /// <summary>PCV02</summary>                  	           
	steam_flow_control_valve_ki											: REAL		:= 0.01;
    /// <summary>PCV02</summary>                  	           
	steam_flow_control_valve_loop_time									: REAL		:= 2000;
    /// <summary>PCV02</summary>                  	           
	steam_flow_control_valve_iband										: REAL		:= 6;
    /// <summary>PCV02</summary>                  	           
	steam_flow_control_valve_base										: INT		:= 13110;
    /// <summary>PCV02</summary>                  	           
	steam_flow_control_valve_base_adjust								: INT		:= 10;
	
	{attribute 'OPC.UA.DA' := '1'}  				                
	{attribute 'OPC.UA.DA.Access' := '1'}  				                
	l1_current_240														: REAL;
	{attribute 'OPC.UA.DA' := '1'}  				                
	{attribute 'OPC.UA.DA.Access' := '1'}  				                
	l1_current_240_error										AT %I*	: BOOL;
	IT1															AT %I*	: INT;
	{attribute 'OPC.UA.DA' := '1'}  				                
	{attribute 'OPC.UA.DA.Access' := '1'}  				                
	l2_current_240														: REAL;
	{attribute 'OPC.UA.DA' := '1'}  				                
	{attribute 'OPC.UA.DA.Access' := '1'}  				                
	l2_current_240_error										AT %I*	: BOOL;
	IT2															AT %I*	: INT;
	{attribute 'OPC.UA.DA' := '1'}  				                
	{attribute 'OPC.UA.DA.Access' := '1'}  				                
	l3_current_240														: REAL;
	{attribute 'OPC.UA.DA' := '1'}  				                
	{attribute 'OPC.UA.DA.Access' := '1'}  				                
	l3_current_240_error										AT %I*	: BOOL;
	IT3															AT %I*	: INT;
	
	{attribute 'OPC.UA.DA' := '1'}  				                
	{attribute 'OPC.UA.DA.Access' := '1'}  				                
	l1_voltage_240														: REAL;
	{attribute 'OPC.UA.DA' := '1'}  				                
	{attribute 'OPC.UA.DA.Access' := '1'}  				                
	l1_voltage_240_error										AT %I*	: BOOL;
	{attribute 'OPC.UA.DA' := '1'}  				                
	VT1															AT %I*	: INT;
	{attribute 'OPC.UA.DA' := '1'}  				                
	l2_voltage_240														: REAL;
	{attribute 'OPC.UA.DA' := '1'}  				                
	{attribute 'OPC.UA.DA.Access' := '1'}  				                
	l2_voltage_240_error										AT %I*	: BOOL;
	{attribute 'OPC.UA.DA' := '1'}  				                
	VT2															AT %I*	: INT;
	{attribute 'OPC.UA.DA' := '1'}  				                
	l3_voltage_240														: REAL;
	{attribute 'OPC.UA.DA' := '1'}  				                
	{attribute 'OPC.UA.DA.Access' := '1'}  				                
	l3_voltage_240_error										AT %I*	: BOOL;
	{attribute 'OPC.UA.DA' := '1'}  				                
	VT3															AT %I*	: INT;
	
	{attribute 'OPC.UA.DA' := '1'}  				                
	{attribute 'OPC.UA.DA.Access' := '1'}  				                
	l1_current_120														: REAL;
	{attribute 'OPC.UA.DA' := '1'}  				                
	{attribute 'OPC.UA.DA.Access' := '1'}  				                
	l1_current_120_error										AT %I*	: BOOL;
	IT4															AT %I*	: INT;
	
	{attribute 'OPC.UA.DA' := '1'}  				                
	{attribute 'OPC.UA.DA.Access' := '1'}  				                
	l1_voltage_120														: REAL;
	{attribute 'OPC.UA.DA' := '1'}  				                
	{attribute 'OPC.UA.DA.Access' := '1'}  				                
	l1_voltage_120_error										AT %I*	: BOOL;
	VT4															AT %I*	: INT;
	
	{attribute 'OPC.UA.DA' := '1'}  				                
	{attribute 'OPC.UA.DA.Access' := '1'}  				                
	l1_current_boiler													: REAL;
	{attribute 'OPC.UA.DA' := '1'}  				                
	{attribute 'OPC.UA.DA.Access' := '1'}  				                
	l1_current_boiler_error										AT %I*	: BOOL;
	IT_boiler_01												AT %I*	: INT;
	{attribute 'OPC.UA.DA' := '1'}  				                
	{attribute 'OPC.UA.DA.Access' := '1'}  				                
	l2_current_boiler													: REAL;
	{attribute 'OPC.UA.DA' := '1'}  				                
	{attribute 'OPC.UA.DA.Access' := '1'}  				                
	l2_current_boiler_error										AT %I*	: BOOL;
	IT_boiler_02												AT %I*	: INT;
	{attribute 'OPC.UA.DA' := '1'}  				                
	{attribute 'OPC.UA.DA.Access' := '1'}  				                
	l3_current_boiler													: REAL;
	{attribute 'OPC.UA.DA' := '1'}  				                
	{attribute 'OPC.UA.DA.Access' := '1'}  				                
	l3_current_boiler_error										AT %I*	: BOOL;
	IT_boiler_03												AT %I*	: INT;
	
	//== Water Scales ====
	  /// <summary>WI01</summary>
	{attribute 'OPC.UA.DA' := '1'}  				                
	{attribute 'OPC.UA.DA.Access' := '1'}  				                
	water_scale_1														: REAL;
    /// <summary>WI01</summary>
	{attribute 'OPC.UA.DA' := '1'}  				                
	{attribute 'OPC.UA.DA.Access' := '1'}  				                
	water_scale_1_error													: BOOL;
    /// <summary>WI01</summary>
	{attribute 'OPC.UA.DA' := '1'}  				                
	_WaterScale1ErrorOff												: BOOL;
    /// <summary>water scale 1</summary>
	WI_01														AT %I*	: INT;
    /// <summary>water scale 1</summary>
	{attribute 'OPC.UA.DA' := '1'}  				                
	{attribute 'OPC.UA.DA.Access' := '1'}  				                
	WI_01_error													AT %I*	: BOOL;
	
	  /// <summary>WI02</summary>
	{attribute 'OPC.UA.DA' := '1'}  				                
	{attribute 'OPC.UA.DA.Access' := '1'}  				                
	water_scale_2														: REAL;
    /// <summary>WI02</summary>
	{attribute 'OPC.UA.DA' := '1'}  				                
	{attribute 'OPC.UA.DA.Access' := '1'}  				                
	water_scale_2_error													: BOOL;
    /// <summary>WI02</summary>
	{attribute 'OPC.UA.DA' := '1'}  				                
	_WaterScale2ErrorOff												: BOOL;
    /// <summary>water scale 2</summary>
	WI_02														AT %I*	: INT;
    /// <summary>water scale 2</summary>
	{attribute 'OPC.UA.DA' := '1'}  				                
	{attribute 'OPC.UA.DA.Access' := '1'}  				                
	WI_02_error													AT %I*	: BOOL;
	
	
		  /// <summary>WI03</summary>
	{attribute 'OPC.UA.DA' := '1'}  				                
	{attribute 'OPC.UA.DA.Access' := '1'}  				                
	water_scale_3														: REAL;
    /// <summary>WI03</summary>
	{attribute 'OPC.UA.DA' := '1'}  				                
	{attribute 'OPC.UA.DA.Access' := '1'}  				                
	water_scale_3_error													: BOOL;
    /// <summary>WI03</summary>
	{attribute 'OPC.UA.DA' := '1'}  				                
	_WaterScale3ErrorOff												: BOOL;
    /// <summary>water scale 3/summary>
	WI_03														AT %I*	: INT;
    /// <summary>water scale 3</summary>
	{attribute 'OPC.UA.DA' := '1'}  				                
	{attribute 'OPC.UA.DA.Access' := '1'}  				                
	WI_03_error													AT %I*	: BOOL;
	
END_VAR

VAR PERSISTENT
	
	/// SCALING
	
    /// <summary>AT02</summary>
	{attribute 'OPC.UA.DA' := '1'}  				                
	product_outlet_co2_low												: REAL;
    /// <summary>AT02</summary>
	{attribute 'OPC.UA.DA' := '1'}  				                
	product_outlet_co2_high												: REAL;
    /// <summary>AT02</summary>
	{attribute 'OPC.UA.DA' := '1'}  				                
	product_outlet_co2_min												: REAL;
    /// <summary>AT02</summary>
	{attribute 'OPC.UA.DA' := '1'}  				                
	product_outlet_co2_offset											: REAL;
	
    /// <summary>AT03</summary>
	{attribute 'OPC.UA.DA' := '1'}  				                
	product_outlet_h2o_low												: REAL;
    /// <summary>AT03</summary>
	{attribute 'OPC.UA.DA' := '1'}  				                
	product_outlet_h2o_high												: REAL;
    /// <summary>AT03</summary>
	{attribute 'OPC.UA.DA' := '1'}  				                
	product_outlet_h2o_min												: REAL;
    /// <summary>AT03</summary>
	{attribute 'OPC.UA.DA' := '1'}  				                
	product_outlet_h2o_offset											: REAL;
	
    /// <summary>FT02</summary>
	{attribute 'OPC.UA.DA' := '1'}  				                
	product_outlet_flow_low												: REAL;
    /// <summary>FT02</summary>
	{attribute 'OPC.UA.DA' := '1'}  				                
	product_outlet_flow_high											: REAL;
    /// <summary>FT02</summary>
	{attribute 'OPC.UA.DA' := '1'}  				                
	product_outlet_flow_min												: REAL;
    /// <summary>FT02</summary>
	{attribute 'OPC.UA.DA' := '1'}  				                
	product_outlet_flow_offset											: REAL;
	
    /// <summary>FT04</summary>
	{attribute 'OPC.UA.DA' := '1'}  				                
	condensate_flow_low													: REAL;
    /// <summary>FT04</summary>
	{attribute 'OPC.UA.DA' := '1'}  				                
	condensate_flow_high												: REAL;
    /// <summary>FT04</summary>
	{attribute 'OPC.UA.DA' := '1'}  				                
	condensate_flow_min													: REAL;
    /// <summary>FT04</summary>
	{attribute 'OPC.UA.DA' := '1'}  				                
	condensate_flow_offset												: REAL;
	
    /// <summary>FT05</summary>
	{attribute 'OPC.UA.DA' := '1'}  				                
	tap_water_feed_flow_low												: REAL;
    /// <summary>FT05</summary>
	{attribute 'OPC.UA.DA' := '1'}  				                
	tap_water_feed_flow_high											: REAL;
    /// <summary>FT05</summary>
	{attribute 'OPC.UA.DA' := '1'}  				                
	tap_water_feed_flow_min												: REAL;
    /// <summary>FT05</summary>
	{attribute 'OPC.UA.DA' := '1'}  				                
	tap_water_feed_flow_offset											: REAL;

    /// <summary>FT06</summary>
	{attribute 'OPC.UA.DA' := '1'}  				                
	steam_flow_low														: REAL;
    /// <summary>FT06</summary>
	{attribute 'OPC.UA.DA' := '1'}  				                
	steam_flow_high														: REAL;
    /// <summary>FT06</summary>
	{attribute 'OPC.UA.DA' := '1'}  				                
	steam_flow_min														: REAL;
    /// <summary>FT06</summary>
	{attribute 'OPC.UA.DA' := '1'}  				                
	steam_flow_offset													: REAL;

    /// <summary>FT07</summary>
	{attribute 'OPC.UA.DA' := '1'}  				                
	vacuum_pump_water_flow_low											: REAL;
    /// <summary>FT07</summary>
	{attribute 'OPC.UA.DA' := '1'}  				                
	vacuum_pump_water_flow_high											: REAL;
    /// <summary>FT07</summary>
	{attribute 'OPC.UA.DA' := '1'}  				                
	vacuum_pump_water_flow_min											: REAL;
    /// <summary>FT07</summary>
	{attribute 'OPC.UA.DA' := '1'}  				                
	vacuum_pump_water_flow_offset										: REAL;
	
    /// <summary>FT08</summary>
	{attribute 'OPC.UA.DA' := '1'}  				                
	condenser_flow_low													: REAL;
    /// <summary>FT08</summary>
	{attribute 'OPC.UA.DA' := '1'}  				                
	condenser_flow_high													: REAL;
    /// <summary>FT08</summary>
	{attribute 'OPC.UA.DA' := '1'}  				                
	condenser_flow_min													: REAL;
    /// <summary>FT08</summary>
	{attribute 'OPC.UA.DA' := '1'}  				                
	condenser_flow_offset												: REAL;
	
    /// <summary>AT-08</summary>                        
	{attribute 'OPC.UA.DA' := '1'}  				            
	weather_wind_speed_low												: REAL;
    /// <summary>AT-08</summary>                        
	{attribute 'OPC.UA.DA' := '1'}  				            
	weather_wind_speed_high												: REAL;
    /// <summary>AT-08</summary>                        
	{attribute 'OPC.UA.DA' := '1'}  				            
	weather_wind_speed_min												: REAL;
    /// <summary>AT-08</summary>                        
	{attribute 'OPC.UA.DA' := '1'}  				            
	weather_wind_speed_offset											: REAL;
	
    /// <summary>LT01</summary>
	{attribute 'OPC.UA.DA' := '1'}  				                
	steam_water_tank_level_low											: REAL;
    /// <summary>LT01</summary>
	{attribute 'OPC.UA.DA' := '1'}  				                
	steam_water_tank_level_high											: REAL;
    /// <summary>LT01</summary>
	{attribute 'OPC.UA.DA' := '1'}  				                
	steam_water_tank_level_min											: REAL;
    /// <summary>LT01</summary>
	{attribute 'OPC.UA.DA' := '1'}  				                
	steam_water_tank_level_offset										: REAL;
	
    /// <summary>LT02</summary>
	{attribute 'OPC.UA.DA' := '1'}  				                
	vacuum_separator_level_low											: REAL;
    /// <summary>LT02</summary>
	{attribute 'OPC.UA.DA' := '1'}  				                
	vacuum_separator_level_high											: REAL;
    /// <summary>LT02</summary>
	{attribute 'OPC.UA.DA' := '1'}  				                
	vacuum_separator_level_min											: REAL;
    /// <summary>LT02</summary>
	{attribute 'OPC.UA.DA' := '1'}  				                
	vacuum_separator_level_offset										: REAL;
	
    /// <summary>PT04</summary>
	{attribute 'OPC.UA.DA' := '1'}  				                
	product_vacuum_pres_low												: REAL;
    /// <summary>PT04</summary>
	{attribute 'OPC.UA.DA' := '1'}  				                
	product_vacuum_pres_high											: REAL;
    /// <summary>PT04</summary>
	{attribute 'OPC.UA.DA' := '1'}  				                
	product_vacuum_pres_min												: REAL;
    /// <summary>PT04</summary>
	{attribute 'OPC.UA.DA' := '1'}  				                
	product_vacuum_pres_offset											: REAL;
	
    /// <summary>PT07</summary>
	{attribute 'OPC.UA.DA' := '1'}  				                
	steam_line_pres_low													: REAL;
    /// <summary>PT07</summary>
	{attribute 'OPC.UA.DA' := '1'}  				                
	steam_line_pres_high												: REAL;
    /// <summary>PT07</summary>
	{attribute 'OPC.UA.DA' := '1'}  				                
	steam_line_pres_min													: REAL;
    /// <summary>PT07</summary>
	{attribute 'OPC.UA.DA' := '1'}  				                
	steam_line_pres_offset												: REAL;
	
    /// <summary>PDT04</summary>
	{attribute 'OPC.UA.DA' := '1'}  				                
	flow_calibration_diff_pres_low										: REAL;
    /// <summary>PDT04</summary>
	{attribute 'OPC.UA.DA' := '1'}  				                
	flow_calibration_diff_pres_high										: REAL;
    /// <summary>PDT04</summary>
	{attribute 'OPC.UA.DA' := '1'}  				                
	flow_calibration_diff_pres_min										: REAL;
    /// <summary>PDT04</summary>
	{attribute 'OPC.UA.DA' := '1'}  				                
	flow_calibration_diff_pres_offset									: REAL;
	
    /// <summary>TT-02</summary>
	{attribute 'OPC.UA.DA' := '1'}  				                
	product_temp_offset													: REAL;
	
    /// <summary>TT-03</summary>
	{attribute 'OPC.UA.DA' := '1'}  				                
	product_vacuum_temp_offset											: REAL;
	
    /// <summary>TT06</summary>
	{attribute 'OPC.UA.DA' := '1'}  				                
	inlet_line_temp_offset												: REAL;
	
    /// <summary>TT10</summary>
	{attribute 'OPC.UA.DA' := '1'}  				                
	vacuum_pump_water_temp_1_offset										: REAL;

    /// <summary>TT11</summary>
	{attribute 'OPC.UA.DA' := '1'}  				                
	vacuum_pump_water_temp_2_offset										: REAL;
	
	
	/// <summary>WI01</summary>
	{attribute 'OPC.UA.DA' := '1'}  				                
	water_scale_1_low													: REAL;
    /// <summary>WI01</summary>
	{attribute 'OPC.UA.DA' := '1'}  				                
	water_scale_1_high													: REAL;
    /// <summary>WI01</summary>
	{attribute 'OPC.UA.DA' := '1'}  				                
	water_scale_1_min													: REAL;
    /// <summary>WI01</summary>
	{attribute 'OPC.UA.DA' := '1'}  				                
	water_scale_1_offset												: REAL;
	
	
	/// <summary>WI02</summary>
	{attribute 'OPC.UA.DA' := '1'}  				                
	water_scale_2_low													: REAL;
    /// <summary>WI02</summary>
	{attribute 'OPC.UA.DA' := '1'}  				                
	water_scale_2_high													: REAL;
    /// <summary>WI02</summary>
	{attribute 'OPC.UA.DA' := '1'}  				                
	water_scale_2_min													: REAL;
    /// <summary>WI02</summary>
	{attribute 'OPC.UA.DA' := '1'}  				                
	water_scale_2_offset												: REAL;
	
	/// <summary>WI03</summary>
	{attribute 'OPC.UA.DA' := '1'}  				                
	water_scale_3_low													: REAL;
    /// <summary>WI03</summary>
	{attribute 'OPC.UA.DA' := '1'}  				                
	water_scale_3_high													: REAL;
    /// <summary>WI03</summary>
	{attribute 'OPC.UA.DA' := '1'}  				                
	water_scale_3_min													: REAL;
    /// <summary>WI02</summary>
	{attribute 'OPC.UA.DA' := '1'}  				                
	water_scale_3_offset												: REAL;
	
	/// SET POINTS
	
	{attribute 'OPC.UA.DA' := '1'}  				                
	SP_adsorb_during_steam_bypass										: BOOL;	
	{attribute 'OPC.UA.DA' := '1'}  				                
	SP_adsorb_during_warmup												: BOOL;
	{attribute 'OPC.UA.DA' := '1'}  				                
	SP_boiler_warmup_duration											: REAL;
	{attribute 'OPC.UA.DA' := '1'}  				                
	SP_condensate_collection_tank_high_level							: REAL;	
	{attribute 'OPC.UA.DA' := '1'}  				                
	SP_condensate_collection_tank_low_level								: REAL;
	{attribute 'OPC.UA.DA' := '1'}  				                
	SP_condensation_collection_tank_emergency_low_level					: REAL;	
	{attribute 'OPC.UA.DA' := '1'}  				                
	SP_duration_to_drain_cooling_and_purge_line_in_module				: REAL;				
	{attribute 'OPC.UA.DA' := '1'}  				                
	SP_duration_to_drain_reactor_set									: REAL;	
	{attribute 'OPC.UA.DA' := '1'}  				                
	SP_evacuation_duration												: REAL;							// PS 11/25/24	
	{attribute 'OPC.UA.DA' := '1'}  				                
	SP_evacuation_ideal_pressure										: REAL;							// PS 11/25/24	
	{attribute 'OPC.UA.DA' := '1'}  				                
	SP_mass_flow_totalizer												: REAL;
	{attribute 'OPC.UA.DA' := '1'}  				                
	SP_maximum_condensate_collection_tank_refill_duration				: REAL;							// PS 08_16_24
	{attribute 'OPC.UA.DA' := '1'}  				                
	SP_maximum_condenser_knockout_drain_duration						: REAL;							// PS 08_22_24
	{attribute 'OPC.UA.DA' := '1'}  				                
	SP_maximum_duration_to_drain_reactor_set							: REAL;	
	{attribute 'OPC.UA.DA' := '1'}  				                
	SP_maximum_inlet_product_vacuum_temperature							: REAL;							// PS 04_30_24	
	{attribute 'OPC.UA.DA' := '1'}  				                
	SP_maximum_reasonable_sorbent_TC_reading							: REAL;
	{attribute 'OPC.UA.DA' := '1'}  				                
	SP_maximum_vacuum_separator_drain_duration							: REAL;							// PS 08_22_24
	{attribute 'OPC.UA.DA' := '1'}  				                
	SP_maximum_vacuum_separator_refill_duration							: REAL;							// PS 08_22_24
	{attribute 'OPC.UA.DA' := '1'}  				                
	SP_minimum_condensate_flow											: REAL;							// PS 08_22_24
	{attribute 'OPC.UA.DA' := '1'}  				                
	SP_minimum_dead_air_line_pressure									: REAL;							// PS 11/27/24
	{attribute 'OPC.UA.DA' := '1'}  				                
	SP_minimum_drainage_pressure										: REAL;	
	{attribute 'OPC.UA.DA' := '1'}  				                
	SP_minimum_reasonable_sorbent_TC_reading							: REAL;
	{attribute 'OPC.UA.DA' := '1'}  				                
	SP_minimum_steam_bypass_duration									: REAL;							// PS 12/2/24
	{attribute 'OPC.UA.DA' := '1'}  				                
	SP_minimum_steam_bypass_flow_rate									: REAL;
	{attribute 'OPC.UA.DA' := '1'}  				                
	SP_minimum_vacuum_cooling_loop_flow									: REAL := 2; 						// PS 11/25/24
	{attribute 'OPC.UA.DA' := '1'}  				                
	SP_max_vacuum_cooling_loop_temp										: REAL := 50;							// PS 11/25/24
	{attribute 'OPC.UA.DA' := '1'}  				                
	SP_minimum_vacuum_liq_seal_flow										: REAL;							// PS 08_13_24
	{attribute 'OPC.UA.DA' := '1'}  				                
	SP_product_condensate_drum_high_level								: REAL;
	{attribute 'OPC.UA.DA' := '1'}  				                
	SP_product_condensate_drum_low_level								: REAL;
	{attribute 'OPC.UA.DA' := '1'}  				                
	SP_reactor_vfd_percent_maximum										: INT;
	{attribute 'OPC.UA.DA' := '1'}  				                
	SP_reactor_vfd_percent_step_duration								: REAL;
	{attribute 'OPC.UA.DA' := '1'}  				                
	SP_reactor_vfd_percent_step_size									: INT;
	{attribute 'OPC.UA.DA' := '1'}  				                
	SP_steam_bypass_duration											: REAL;
	{attribute 'OPC.UA.DA' := '1'}  				                
	SP_steam_bypass_immediately_after_warm_up							: BOOL;
	{attribute 'OPC.UA.DA' := '1'}  				                
	SP_steam_bypass_temperature											: REAL;
	{attribute 'OPC.UA.DA' := '1'}  				                
	SP_steam_bypass_vacuum_pressure										: REAL;
	{attribute 'OPC.UA.DA' := '1'}  				                
	SP_target_boiler_pressure											: REAL;
	{attribute 'OPC.UA.DA' := '1'}  				                
	SP_vacuum_pres_control_valve										: REAL;
	{attribute 'OPC.UA.DA' := '1'}  				                
	SP_vacuum_separator_level_emergency_high							: REAL;							// PS 08_13_24									
	{attribute 'OPC.UA.DA' := '1'}  				                
	SP_vacuum_separator_level_emergency_low								: REAL;							// PS 08_13_24									
	{attribute 'OPC.UA.DA' := '1'}  				                
	SP_vacuum_separator_level_high										: REAL;							// PS 08_22_24									
	{attribute 'OPC.UA.DA' := '1'}  				                
	SP_vacuum_separator_level_mid										: REAL;							// PS 08_22_24									
	{attribute 'OPC.UA.DA' := '1'}  				                
	SP_vacuum_separator_level_low										: REAL;							// PS 08_22_24	
	{attribute 'OPC.UA.DA' := '1'}  				                
	SP_waste_water_tank_weight_full										: REAL;										
	{attribute 'OPC.UA.DA' := '1'}  				                
	SP_waste_water_tank_weight_empty									: REAL;	
	{attribute 'OPC.UA.DA' := '1'}  				                
	SP_steam_water_tank_weight_full										: REAL;										
	{attribute 'OPC.UA.DA' := '1'}  				                
	SP_steam_water_tank_weight_empty									: REAL;	
	
	
	
    /// <summary>PCV01</summary>
	vacuum_pres_control_valve_setpoint									: REAL;
	
END_VAR

// Theseus - P_U01
// Rev 1.0 - December 2, 2024

A_IO_Points();
A_PIDs();
A_MovingAverage();
A02_WarmUp();
A03_Steam_Bypass();
A08_Shutdown();
A09_Pressure_Drop_Test();
P_U01.shutdown_process													:= FALSE;

IF LEFT(gsCycleMode, 1) = '0' THEN
	IF gsCycleMode = '02' THEN
		i2Step															:= 1;
	ELSIF gsCycleMode = '03' THEN
		i3Step															:= 1;
	ELSIF gsCycleMode = '08' THEN
		i8Step															:= 1;
	ELSIF gsCycleMode = '09' THEN
		i9Step															:= 1;
	END_IF
	gsCycleMode															:= '';
END_IF

IF tonWriteData.Q OR P_U01.write_persistent_data THEN
	P_U01.write_persistent_data											:= FALSE;
	bWriteData															:= TRUE;
ELSIF NOT fbWriteData.BUSY THEN
	bWriteData															:= FALSE;
END_IF

fbWriteData(	NETID													:= '',
				PORT													:= 851,
				START													:= bWriteData,
				TMOUT													:= T#5S);

tonTimer(IN:= bTimer, PT:= REAL_TO_TIME(rTime));
tonAdsorptionTimer(IN:= bAdsorptionTimer, PT:= REAL_TO_TIME(P_M01.SP_adsorption_duration * _MINUTES));
tonWriteData(IN:= NOT bWriteData, PT:= T#30M);

// Water Scales
fb_WaterScales_In ( 
			i_value := water_scale_1 + water_scale_2,
			io_reset	:= water_scales_reset,
			o_change_value => water_scales_in_delta,
			o_change_rate => water_scales_in_rate
			);
			
fb_WaterScales_Out ( 
			i_value := water_scale_3,
			io_reset	:= water_scales_reset,
			o_change_value => water_scales_out_delta,
			o_change_rate => water_scales_out_rate
			);
		
IF water_scales_reset THEN
	water_scales_reset := FALSE;
END_IF

// Water Scales Capapcity Desorption 
condenser_tank_capacity := SP_waste_water_tank_weight_full - SP_waste_water_tank_weight_empty;
steam_delivery_tank_capacity := SP_steam_water_tank_weight_full - SP_steam_water_tank_weight_empty;
condenser_tank_room_before_full	:= SP_waste_water_tank_weight_full - water_scale_3;
steam_delivery_tank_before_empty := (water_scale_1 + water_scale_2) -  SP_steam_water_tank_weight_empty;

ACTION A_IO_Points:
// Theseus - A_IO_Points
// Rev 1.0 - November 26, 2024

interlock_condenser_steam_or_status										:= interlock_condenser_steam_or;
interlock_hot_reactor_condenser_or_status								:= interlock_hot_reactor_condenser_or;
interlock_no_steam_unevacuated_reactor_or_status						:= interlock_no_steam_unevacuated_reactor_or;
interlock_cooling_with_vacuum_or_status									:= interlock_cooling_with_vacuum_or;
interlock_separator_water_level_with_vacuum_or_status					:= interlock_separator_water_level_with_vacuum_or;
interlock_cooling_loop_flow_with_vacuum_or_status						:= interlock_cooling_loop_flow_with_vacuum_or;
interlock_condensate_tank_level_for_steam_or_status						:= interlock_condensate_tank_level_for_steam_or;
interlock_hot_sorbent_for_repressurization_or_status					:= interlock_hot_sorbent_for_repressurization_or;
interlock_reactor_over_safe_pressure_limit_or_status					:= interlock_reactor_over_safe_pressure_limit_or;
interlock_reactor_over_safe_temperature_limit_or_status					:= interlock_reactor_over_safe_temperature_limit_or;
interlock_repressurization_valve_with_steam_or_status					:= interlock_repressurization_valve_with_steam_or;
interlock_door_open_with_steam_flow_or_status							:= interlock_door_open_with_steam_flow_or;
interlock_door_open_with_reactor_vacuum_or_status						:= interlock_door_open_with_reactor_vacuum_or;
interlock_co2_adsorption_or_status										:= interlock_co2_adsorption_or;
interlock_condensate_pump_or_status										:= interlock_condensate_pump_or;
condenser_knockout_drain_or_on_status									:= condenser_knockout_drain_or_on;
condenser_knockout_drain_or_off_status									:= condenser_knockout_drain_or_off;
vacuum_separator_drain_or_on_status										:= vacuum_separator_drain_or_on;
vacuum_separator_drain_or_off_status									:= vacuum_separator_drain_or_off;
reactor_drain_or_on_status												:= reactor_drain_or_on;
reactor_drain_or_off_status												:= reactor_drain_or_off;

// Interlock 5
cooling_with_vacuum_interlock											:= NOT vacuum_liquid_loop_fan OR NOT vacuum_liquid_pump;
bCondition1																:= NOT interlock_cooling_with_vacuum_or AND cooling_with_vacuum_interlock;

// Interlock 6
separator_water_level_with_vacuum_interlock								:= vacuum_separator_level < SP_vacuum_separator_level_emergency_low OR vacuum_separator_level > SP_vacuum_separator_level_emergency_high;
bCondition2																:= NOT interlock_separator_water_level_with_vacuum_or AND separator_water_level_with_vacuum_interlock;

// Interlock 7
cooling_loop_flow_with_vacuum_interlock									:= vacuum_pump AND vacuum_pump_water_flow < SP_minimum_vacuum_liq_seal_flow;
tonVacuumInterlock(IN:= cooling_loop_flow_with_vacuum_interlock, PT:= T#5S);
bCondition3																:= NOT interlock_cooling_loop_flow_with_vacuum_or AND tonVacuumInterlock.Q;

IF bCondition1 OR bCondition2 OR bCondition3 THEN
	vacuum_pump															:= FALSE;
END_IF
IF bCondition2 THEN
	vacuum_pump_inlet_valve												:= FALSE;
	vacuum_pump_bypass_valve											:= FALSE;
	dead_air_inlet_valve												:= FALSE;
	product_line_ambient_valve											:= INT_TO_BOOL(eAmbient);
END_IF

// Interlock 8
condensate_tank_level_for_steam_interlock								:= steam_water_tank_level < SP_condensation_collection_tank_emergency_low_level;
IF NOT interlock_condensate_tank_level_for_steam_or AND condensate_tank_level_for_steam_interlock THEN
	boiler_package														:= FALSE;
	steam_water_pump													:= FALSE;
	steam_flow_control_valve											:= _CLOSED;
END_IF

gbDrainageOn															:= (drainage_on AND NOT drainage_function_off_or) OR drainage_function_on_or;

// Interlock 9
hot_sorbent_for_repressurization_interlock								:= P_M01.rs1.sorbent_high_temp >= P_M01.SP_maximum_target_sorbent_temperature_to_repressurize;
bCondition1																:= NOT interlock_hot_sorbent_for_repressurization_or AND hot_sorbent_for_repressurization_interlock;
 
// Interlock 13
P_U01.repressurization_valve_with_steam_interlock						:= NOT P_U01.steam_flow_control_valve_closed;
bCondition2																:= NOT P_U01.interlock_repressurization_valve_with_steam_or AND P_U01.repressurization_valve_with_steam_interlock;

gbRepresValves															:= NOT bCondition1 AND NOT bCondition2;

// Vacuum Separator
IF (gbDrainageOn OR vacuum_separator_drain_or_on) AND NOT vacuum_separator_drain_or_off THEN
	// Fill
	tonVacuumSeparatorFill(IN:= tap_water_feed_valve AND NOT bVacuumSeparatorFillError, PT:= REAL_TO_TIME(SP_maximum_vacuum_separator_refill_duration * _MINUTES));
	IF tonVacuumSeparatorFill.Q THEN
		tap_water_feed_valve											:= FALSE;
		bVacuumSeparatorFillError										:= TRUE;
		P_Alarms.M_Add_Alarm(_U01, gsVacuumSeparatorFillError, gsMessageTBD);
	ELSIF vacuum_separator_level < SP_vacuum_separator_level_low  AND NOT bVacuumSeparatorFillError THEN
		tap_water_feed_valve											:= TRUE;
	ELSIF vacuum_separator_level > SP_vacuum_separator_level_mid THEN
		tap_water_feed_valve											:= FALSE;
		bVacuumSeparatorFillError										:= FALSE;
	END_IF
	// Drain
//	tonVacuumSeparatorDrain(IN:= separator_drain_valve AND NOT bVacuumSeparatorDrainError, PT:= REAL_TO_TIME(SP_maximum_vacuum_separator_drain_duration * _MINUTES));
	IF tonVacuumSeparatorFill.Q THEN
		separator_drain_valve											:= FALSE;
		vacuum_separator_drain_pump										:= FALSE;
		bVacuumSeparatorDrainError										:= TRUE;
		P_Alarms.M_Add_Alarm(_U01, gsVacuumSeparatorDrainError, gsMessageTBD);
	ELSIF vacuum_separator_level >= SP_vacuum_separator_level_high THEN
		separator_drain_valve											:= TRUE;
		vacuum_separator_drain_pump										:= TRUE;
	ELSIF vacuum_separator_level < SP_vacuum_separator_level_mid THEN
		separator_drain_valve											:= FALSE;
		vacuum_separator_drain_pump										:= FALSE;
		bVacuumSeparatorDrainError										:= FALSE;
	END_IF
END_IF
rtrigVacuumSeparator(CLK:= NOT gbDrainageOn AND NOT vacuum_separator_drain_or_on AND NOT vacuum_separator_drain_or_off);
IF rtrigVacuumSeparator.Q THEN
	tap_water_feed_valve												:= FALSE;
	separator_drain_valve												:= FALSE;
	vacuum_separator_drain_pump											:= FALSE;
END_IF

// Condenser Knockout drainage
IF (gbDrainageOn OR condenser_knockout_drain_or_on) AND NOT condenser_knockout_drain_or_off THEN
	IF gbCondenserKODrainageOn THEN
//		tonCondenserKODrain(IN:= NOT bCondenserKnockoutError AND (product_condensate_drum_lsh OR product_condensate_drum_lsl), PT:= REAL_TO_TIME(SP_maximum_condenser_knockout_drain_duration * _MINUTES));
		IF tonCondenserKODrain.Q AND P_M01.rs1.reactor_condensate_flow < SP_minimum_condensate_flow THEN
			bCondenserKnockoutError										:= TRUE;
			knockout_drain_valve										:= FALSE;
			steam_flow_control_valve									:= _CLOSED;
			P_Alarms.M_Add_Alarm(_U01, gsCondenserKODrainageError, gsMessageTBD);
		ELSIF product_condensate_drum_lsh THEN
			knockout_drain_valve										:= TRUE;
		ELSIF NOT product_condensate_drum_lsh AND NOT product_condensate_drum_lsl THEN
			knockout_drain_valve										:= FALSE;
		END_IF
	ELSE
		knockout_drain_valve											:= FALSE;
	END_IF
END_IF
rtrigKODrainValve(CLK:= NOT gbDrainageOn AND NOT condenser_knockout_drain_or_on AND NOT condenser_knockout_drain_or_off);
IF rtrigKODrainValve.Q THEN
	knockout_drain_valve												:= FALSE;
END_IF

fb_adsorp_product_wastewater
	( i_execute := condenser_knockout_drain_adsorption_on,
	  i_value := P_U01.water_scale_3,
	  i_time := 30,
	  i_threshold := 1);
	  
IF condenser_knockout_drain_adsorption_on THEN
	IF NOT fb_adsorp_product_wastewater.o_below_threshold THEN
		knockout_drain_valve											:= TRUE;
	ELSIF fb_adsorp_product_wastewater.o_below_threshold OR fb_adsorp_product_wastewater.o_timeout THEN
		knockout_drain_valve											:= FALSE;
		condenser_knockout_drain_adsorption_on 							:= FALSE;
	END_IF
END_IF


IF NOT interlock_condensate_pump_or THEN
	condensate_pump														:= knockout_drain_valve OR gbCondensateValve;
END_IF

// Interlock 2
condenser_steam_interlock												:= NOT steam_flow_control_valve_closed AND (P_M01.rs1.steam_bypass_valve_open OR P_M01.rs1.product_iso_valve_open);
IF NOT interlock_condenser_steam_or AND condenser_steam_interlock THEN
	condenser_pump														:= TRUE;
	condenser_fan														:= TRUE;
END_IF

B_01																	:= boiler_package;
boiler_package_cmd_status												:= B_01;

P_01																	:= steam_water_pump;
steam_water_pump_cmd_status												:= P_01;

P_02																	:= vacuum_pump;
vacuum_pump_cmd_status													:= P_02;

P_03																	:= condensate_pump;
condensate_pump_cmd_status												:= P_03;

P_04																	:= condenser_pump;
condenser_pump_cmd_status												:= P_04;

P_05																	:= vacuum_liquid_pump;
vacuum_liquid_pump_cmd_status											:= P_05;

P_06																	:= vacuum_separator_drain_pump;
vacuum_separator_drain_pump_cmd_status									:= P_06;

E_01																	:= condenser_fan;
condenser_fan_cmd_status												:= E_01; 

X_01																	:= vacuum_liquid_loop_fan;
vacuum_liquid_loop_fan_cmd_status										:= X_01;

product_outlet_co2														:= F_AnalogIn(AT_02, product_outlet_co2_low, product_outlet_co2_high, product_outlet_co2_min, product_outlet_co2_offset);
product_outlet_co2_error												:= AT_02_error AND NOT _ProductOutletCO2ErrorOff;
bProductOutletCo2Error													:= P_Alarms.M_Check_Error(product_outlet_co2_error, bProductOutletCo2Error, _U01, gsProductOutletCo2SensorError, gsProcessCannotRun);

product_outlet_h2o														:= F_AnalogIn(AT_03, product_outlet_h2o_low, product_outlet_h2o_high, product_outlet_h2o_min, product_outlet_h2o_offset);
product_outlet_h2o_error												:= AT_03_error AND NOT _ProductOutletH2OErrorOff;
bProductOutletH2oError													:= P_Alarms.M_Check_Error(product_outlet_h2o_error, bProductOutletH2oError, _U01, gsProductOutletH2oSensorError, gsProcessCannotRun);

product_outlet_flow														:= F_AnalogIn(FT_02, product_outlet_flow_low, product_outlet_flow_high, product_outlet_flow_min, product_outlet_flow_offset);
product_outlet_flow_error												:= product_outlet_flow_error AND NOT _ProductOutletFlowErrorOff;
bProductOutletFlowError													:= P_Alarms.M_Check_Error(product_outlet_flow_error, bProductOutletFlowError, _U01, gsProductOutletFlowSensorError, gsProcessCannotRun);

condensate_flow															:= F_AnalogIn(FT_04, condensate_flow_low, condensate_flow_high, condensate_flow_min, condensate_flow_offset);
condensate_flow_error													:= FT_04_error AND NOT _CondensateFlowErrorOff;
bCondensateFlowError													:= P_Alarms.M_Check_Error(condensate_flow_error, bCondensateFlowError, _U01, gsCondensateFlowSensorError, gsProcessCannotRun);
	
tap_water_feed_flow														:= F_AnalogIn(FT_05, tap_water_feed_flow_low, tap_water_feed_flow_high, tap_water_feed_flow_min, tap_water_feed_flow_offset);
tap_water_feed_flow_error												:= FT_05_error AND NOT _TapWaterFeedFlowErrorOff;
bWaterFeedFlowError														:= P_Alarms.M_Check_Error(tap_water_feed_flow_error, bWaterFeedFlowError, _U01, gsTapWaterFeedFlowSensorError, gsProcessCannotRun);

steam_flow																:= F_AnalogIn(FT_06, steam_flow_low, steam_flow_high, steam_flow_min, steam_flow_offset);
steam_flow_error														:= FT_06_error AND NOT _SteamFlowErrorOff;
bSteamFlowError															:= P_Alarms.M_Check_Error(steam_flow_error, bSteamFlowError, _U01, gsTapWaterFeedFlowSensorError, gsProcessCannotRun);

vacuum_pump_water_flow													:= F_AnalogIn(FT_07, vacuum_pump_water_flow_low, vacuum_pump_water_flow_high, vacuum_pump_water_flow_min, vacuum_pump_water_flow_offset);
vacuum_pump_water_flow_error											:= FT_07_error AND NOT _VacuumPumpWaterFlowErrorOff;
bVacuumPumpWaterFlowError												:= P_Alarms.M_Check_Error(vacuum_pump_water_flow_error, bVacuumPumpWaterFlowError, _U01, gsVacuumPumpWaterFlowSensorError, gsProcessCannotRun);
	
condenser_flow															:= F_AnalogIn(FT_08, condenser_flow_low, condenser_flow_high, condenser_flow_min, condenser_flow_offset);
condenser_flow_error													:= FT_08_error AND NOT _CondenserFlowErrorOff;
bCondenserFlowError														:= P_Alarms.M_Check_Error(condenser_flow_error, bCondenserFlowError, _U01, gsCondenserFlowSensorError, gsProcessCannotRun);
	
steam_water_tank_level													:= F_AnalogIn(LT_01, steam_water_tank_level_low, steam_water_tank_level_high, steam_water_tank_level_min, steam_water_tank_level_offset);
steam_water_tank_level_error											:= LT_01_error AND NOT _SteamWaterTankLevelErrorOff;
bSteamWaterTankLevelError												:= P_Alarms.M_Check_Error(steam_water_tank_level_error, bSteamWaterTankLevelError, _U01, gsSteamWaterTankLevelSensorError, gsProcessCannotRun);
	
vacuum_separator_level													:= F_AnalogIn(LT_02, vacuum_separator_level_low, vacuum_separator_level_high, vacuum_separator_level_min, vacuum_separator_level_offset);
vacuum_separator_level_error											:= LT_02_error AND NOT _VacuumSeparatorLevelErrorOff;
bVacuumSeparatorLevelError												:= P_Alarms.M_Check_Error(vacuum_separator_level_error, bVacuumSeparatorLevelError, _U01, gsVacuumSeparatorLevelSensorError, gsProcessCannotRun);
	
product_vacuum_pres														:= F_AnalogIn(PT_04, product_vacuum_pres_low, product_vacuum_pres_high, product_vacuum_pres_min, product_vacuum_pres_offset);
product_vacuum_pres_error												:= PT_04_error AND NOT _ProductVacuumPresErrorOff;
bProductVacuumPresError													:= P_Alarms.M_Check_Error(product_vacuum_pres_error, bProductVacuumPresError, _U01, gsProductVacuumPresSensorError, gsProcessCannotRun);

steam_line_pres															:= F_AnalogIn(PT_07, steam_line_pres_low, steam_line_pres_high, steam_line_pres_min, steam_line_pres_offset);
steam_line_pres_error													:= PT_07_error AND NOT _SteamLinePresErrorOff;
bSteamLinePresError														:= P_Alarms.M_Check_Error(steam_line_pres_error, bSteamLinePresError, _U01, gsSteamLinePresSensorError, gsProcessCannotRun);

flow_calibration_diff_pres												:= F_AnalogIn(PDT_04, flow_calibration_diff_pres_low, flow_calibration_diff_pres_high, flow_calibration_diff_pres_min, flow_calibration_diff_pres_offset);
flow_calibration_diff_pres_error										:= PDT_04_error AND NOT _FlowCalibrationDiffPresErrorOff;
bFlowCalibrationDiffPresError											:= P_Alarms.M_Check_Error(flow_calibration_diff_pres_error, bFlowCalibrationDiffPresError, _U01, gsFlowCalibrationDiffPresSensorError, gsProcessCannotRun);


water_scale_1															:= F_AnalogIn(WI_01, water_scale_1_low, water_scale_1_high, water_scale_1_min, water_scale_1_offset);
water_scale_1_error														:= WI_01_error AND NOT _WaterScale1ErrorOff;
bWaterScale1Error														:= P_Alarms.M_Check_Error(water_scale_1_error, bWaterScale1Error, _U01, gsWaterScale1SensorError, gsWarning); 
	
water_scale_2															:= F_AnalogIn(WI_02, water_scale_2_low, water_scale_2_high, water_scale_2_min, water_scale_2_offset);
water_scale_2_error														:= WI_02_error AND NOT _WaterScale2ErrorOff;
bWaterScale2Error														:= P_Alarms.M_Check_Error(water_scale_2_error, bWaterScale2Error, _U01, gsWaterScale1SensorError, gsWarning); 

water_scale_3															:= F_AnalogIn(WI_03, water_scale_3_low, water_scale_3_high, water_scale_3_min, water_scale_3_offset);
water_scale_3_error														:= WI_03_error AND NOT _WaterScale3ErrorOff;
bWaterScale3Error														:= P_Alarms.M_Check_Error(water_scale_3_error, bWaterScale3Error, _U01, gsWaterScale1SensorError, gsWarning);

product_temp															:= F_Temperature(TT_02, product_temp_offset);
product_temp_error														:= TT_02_error AND NOT _ProductTempErrorOff;
bProductTempError														:= P_Alarms.M_Check_Error(product_temp_error, bProductTempError, _U01, gsProductTempSensorError, gsProcessCannotRun);

product_vacuum_temp														:= F_Temperature(TT_03, product_vacuum_temp_offset);
product_vacuum_temp_error												:= TT_03_error AND NOT _ProductVacuumTempOff;
bProductVacuumTempError													:= P_Alarms.M_Check_Error(product_vacuum_temp_error, bProductVacuumTempError, _U01, gsProductVacuumTempSensorError, gsProcessCannotRun);
	
inlet_line_temp															:= F_Temperature(TT_06, inlet_line_temp_offset);
inlet_line_temp_error													:= TT_06_error AND NOT _InletLineTempErrorOff;
bInletLineTempError														:= P_Alarms.M_Check_Error(inlet_line_temp_error, bInletLineTempError, _U01, gsInletLineTempSensorError, gsProcessCannotRun);

vacuum_pump_water_temp_1												:= F_Temperature(TT_10, vacuum_pump_water_temp_1_offset);
vacuum_pump_water_temp_1_error											:= TT_10_error AND NOT _VacuumPumpWaterTemp1ErrorOff;
bVacuumPumpWaterTemp1Error												:= P_Alarms.M_Check_Error(vacuum_pump_water_temp_1_error, bVacuumPumpWaterTemp1Error, _U01, gsVacuumPumpWaterTemp1SensorError, gsProcessCannotRun);

vacuum_pump_water_temp_2												:= F_Temperature(TT_11, vacuum_pump_water_temp_2_offset);
vacuum_pump_water_temp_2_error											:= TT_11_error AND NOT _VacuumPumpWaterTemp2ErrorOff;

IF bCloseXVValves THEN
	vacuum_pump_inlet_valve												:= FALSE;
	vacuum_pump_bypass_valve											:= FALSE;
	knockout_drain_valve												:= FALSE;
	dead_air_inlet_valve												:= FALSE;
	separator_drain_valve												:= FALSE;
	bCloseXVValves														:= FALSE;
END_IF

XV_03																	:= 	vacuum_pump_inlet_valve;
vacuum_pump_inlet_valve_open_cmd_status									:= vacuum_pump_inlet_valve;
vacuum_pump_inlet_valve_clear											:= F_ValveClear(vacuum_pump_inlet_valve, vacuum_pump_inlet_valve_open, vacuum_pump_inlet_valve_closed);

XV_04																	:= vacuum_pump_bypass_valve;
vacuum_pump_bypass_valve_open_cmd_status								:= XV_04;
vacuum_pump_bypass_valve_clear											:= F_ValveClear(vacuum_pump_bypass_valve, vacuum_pump_bypass_valve_open, vacuum_pump_bypass_valve_closed);

XV_06																	:= knockout_drain_valve;
knockout_drain_valve_open_cmd_status									:= XV_06;
knockout_drain_valve_clear												:= F_ValveClear(knockout_drain_valve, knockout_drain_valve_open, knockout_drain_valve_closed);

XV_10																	:= dead_air_inlet_valve;
dead_air_inlet_valve_open_cmd_status									:= dead_air_inlet_valve;
dead_air_inlet_valve_clear												:= F_ValveClear(dead_air_inlet_valve, dead_air_inlet_valve_open, dead_air_inlet_valve_closed);

XV_11																	:= product_line_ambient_valve;
product_line_ambient_valve_cmd_status									:= XV_11;
product_line_ambient_valve_clear										:= F_ValveClear(product_line_ambient_valve, product_line_ambient_valve_ambient,product_line_ambient_valve_product);

XV_12																	:= tap_water_feed_valve;
tap_water_feed_valve_cmd_status											:= XV_12;

XV_13																	:= separator_drain_valve;
separator_drain_valve_open_cmd_status									:= XV_13;
separator_drain_valve_clear												:= F_ValveClear(separator_drain_valve, separator_drain_valve_open, separator_drain_valve_closed);

XV_14																	:= steam_water_reservoir_valve;
steam_water_reservoir_valve_cmd_status									:= XV_14;

fb_Vacuum_Pres_Control_Valve_PI(		Setpoint						:= vacuum_pres_control_valve_setpoint,
										Control							:= product_vacuum_pres,
										Error							:= vacuum_pres_control_valve_position_error,
										Reverse							:= FALSE,
										Kp								:= vacuum_pres_control_valve_kp,           
										Ki								:= vacuum_pres_control_valve_ki,           
										BaseAdjust						:= vacuum_pres_control_valve_base_adjust,  
										LoopTime						:= vacuum_pres_control_valve_loop_time,    
										IBand							:= vacuum_pres_control_valve_iband,        
										Base							:= vacuum_pres_control_valve_base,         
										Mode							:= vacuum_pres_control_valve_mode,
										Input							:= vacuum_pres_control_valve,
										Mode_Out						=> vacuum_pres_control_valve_current_mode, 
										Output							=> PCV_01);

vacuum_pres_control_valve_position										:= INT_TO_REAL(PCV_01_position) / _PERCENT_FACTOR; 
vacuum_pres_control_valve_open											:= vacuum_pres_control_valve_position >= _VALVE_OPEN;
vacuum_pres_control_valve_closed										:= vacuum_pres_control_valve_position < _VALVE_CLOSED;

fb_Steam_Flow_Control_Valve_PI(			Setpoint						:= steam_flow_control_valve_setpoint,
										Control							:= ,
										Error							:= steam_flow_control_valve_position_error,
										Reverse							:= FALSE,
										Kp								:= steam_flow_control_valve_kp,           
										Ki								:= steam_flow_control_valve_ki,           
										BaseAdjust						:= steam_flow_control_valve_base_adjust,  
										LoopTime						:= steam_flow_control_valve_loop_time,    
										IBand							:= steam_flow_control_valve_iband,        
										Base							:= steam_flow_control_valve_base,         
										Mode							:= steam_flow_control_valve_mode,
										Input							:= steam_flow_control_valve,
										Mode_Out						=> steam_flow_control_valve_current_mode, 
										Output							=> PCV_02);

steam_flow_control_valve_position										:= INT_TO_REAL(PCV_02_position) / _PERCENT_FACTOR; 
steam_flow_control_valve_open											:= steam_flow_control_valve_position >= _VALVE_OPEN;
steam_flow_control_valve_closed											:= steam_flow_control_valve_position < _VALVE_CLOSED;

// ignore if < 2 Amps
l1_current_240															:= SEL(IT1 > _CURRENT_240_FACTOR * 2,0,F_IEConvert(IT1, _CURRENT_240_FACTOR));
l2_current_240															:= SEL(IT2 > _CURRENT_240_FACTOR * 2,0,F_IEConvert(IT2, _CURRENT_240_FACTOR));
l3_current_240															:= SEL(IT3 > _CURRENT_240_FACTOR * 2,0,F_IEConvert(IT3, _CURRENT_240_FACTOR));
l1_voltage_240															:= F_IEConvert(VT1, _VOLTAGE_240_FACTOR);
l2_voltage_240															:= F_IEConvert(VT2, _VOLTAGE_240_FACTOR);
l3_voltage_240															:= F_IEConvert(VT3, _VOLTAGE_240_FACTOR);

// Ignore if < 1 Amp
l1_current_120															:= SEL(IT4 > _CURRENT_120_FACTOR ,0,F_IEConvert(IT4, _CURRENT_120_FACTOR));
l1_voltage_120															:= F_IEConvert(VT4, _VOLTAGE_120_FACTOR);

// Boiler - ignore noise if < 5A = 400 counts

l1_current_boiler := SEL(IT_boiler_01 > 400, 0, F_IEConvert(IT_boiler_01, _CURRENT_BOILER_FACTOR));  // double coiled 
l2_current_boiler := SEL(IT_boiler_02 > 400, 0, F_IEConvert(IT_boiler_02, _CURRENT_BOILER_FACTOR));  // double coiled 
l3_current_boiler := SEL(IT_boiler_03 > 400, 0, F_IEConvert(IT_boiler_03, _CURRENT_BOILER_FACTOR));  // double coiled 

//boiler_ready														:= NOT boiler_outlet_pres_error AND boiler_outlet_pres > SP_target_boiler_pressure AND boiler_package;
//boiler_ready															:= boiler_ready;

tonBoilerCheck(IN:= warmup_complete AND NOT boiler_ready, PT:= _TIMEOUT_WARMUP_RESET);
IF tonBoilerCheck.Q THEN
	warmup_complete														:= FALSE;
END_IF

// These Utility errors prevent any new automated cycles from running
utility_error		:= '';
//utility_error															:= SEL(NOT boiler_ready, '', gsBoilerError);
utility_error															:= SEL(bProductVacuumPresError, utility_error, gsProductVacuumPresSensorError);
//utility_error															:= SEL(bProductOutletCo2Error, utility_error, gsProductOutletCo2SensorError);
//utility_error															:= SEL(bInletLineTempError, utility_error, gsInletLineTempSensorError);
//utility_error															:= SEL(bSteamWaterTankLevelError, utility_error, gsSteamWaterTankLevelSensorError);
utility_error															:= SEL(bVacuumSeparatorLevelError, utility_error, gsVacuumSeparatorLevelSensorError);
utility_error															:= SEL(bVacuumPumpWaterFlowError, utility_error, gsVacuumPumpWaterFlowSensorError);
utility_error															:= SEL(bVacuumPumpWaterTemp1Error, utility_error, gsVacuumPumpWaterTemp1SensorError);
//utility_error															:= SEL(bFlowCalibrationDiffPresError, utility_error, gsFlowCalibrationDiffPresSensorError);
//utility_error															:= SEL(bProductOutletH2oError, utility_error, gsProductOutletH2oSensorError);
//utility_error															:= SEL(bProductTempError, utility_error, gsProductTempSensorError);
//utility_error															:= SEL(bProductVacuumTempError, utility_error, gsProductVacuumTempSensorError);
//utility_error															:= '';

//sUtilityError															:= utility_error; // - TO BE ENABLED
END_ACTION

ACTION A_MovingAverage:
(*
moving_avg_params.nSamplesToFilter := 2;
moving_avg_params.tCtrlCycleTime := T#1000MS;
moving_avg_params.tTaskCycleTime := T#10MS;
moving_avg_params.pWorkArray_ADR := ADR(moving_avg_array);
moving_avg_params.nWorkArray_SIZEOF := SIZEOF(moving_avg_array);

moving_avg_in_sim_timer ( IN := NOT moving_avg_in_sim_timer.Q, PT := T#1000MS);

IF moving_avg_in_sim_timer.Q THEN 
	moving_avg_in := moving_avg_in + 1;
	IF moving_avg_in = 100 THEN
		moving_avg_in := 0;
	END_IF
END_IF

fb_MovingAverage(
	fIn:= moving_avg_in , 
	fManSyncValue:= , 
	bSync:= , 
	eMode:= E_CTRL_MODE.eCTRL_MODE_ACTIVE, 
	bHold:= , 
	fOut=> moving_avg_out, 
	eState=> , 
	eErrorId=> , 
	bError=> , 
	stParams:= moving_avg_params);
*)

fbMovingAverage(
	i_number_of_samples := 5,
	i_sample_time := 1000);
END_ACTION

ACTION A_PIDs:
// Steam valve

steam_valve_pid_params.tCtrlCycleTime := T#1000MS;
steam_valve_pid_params.tTaskCycleTime := T#10MS;
steam_valve_pid_params.fKp := steam_valve_pid_kp ;
steam_valve_pid_params.tTn := steam_valve_pid_tn;
steam_valve_pid_params.tTv := steam_valve_pid_tv;
steam_valve_pid_params.tTd := T#0MS;
steam_valve_pid_params.fOutMaxLimit := 100;
steam_valve_pid_params.fOutMinLimit := 0;

steam_valve_pid(
	fSetpointValue	:= steam_valve_pid_sp_value, 
	fActualValue	:= steam_valve_pid_actual_value, 
	fManSyncValue	:= steam_valve_pid_manual_sp, 
	bSync			:= FALSE, 
	eMode			:= steam_valve_pid_mode , 
	bHold:= , 
	fOut			=> steam_valve_pid_out , 
	bARWactive=> , 
	eState=> , 
	eErrorId=> , 
	bError=> , 
	stParams		:= steam_valve_pid_params);


steam_valve_pid_simulate_timer( IN := NOT steam_valve_pid_simulate_timer.Q, PT := T#10MS);
IF steam_valve_pid_simulate_timer.Q AND steam_valve_pid.eMode = E_CTRL_MODE.eCTRL_MODE_ACTIVE THEN
	//steam_valve_pid_actual_value := steam_valve_pid_actual_value * 0.8 + steam_valve_pid_out * 0.01;
	//steam_valve_pid_actual_value := steam_valve_pid_actual_value + ((steam_valve_pid_sp_value - steam_valve_pid_actual_value)/1.2) + 0.1; 
	steam_valve_pid_actual_value := steam_valve_pid_actual_value * 0.995 + steam_valve_pid_out * 0.01;
END_IF
(*	
IF steam_valve_pid.eMode = E_CTRL_MODE.eCTRL_MODE_MANUAL  AND (steam_valve_pid_sp_value <= 0) THEN
	steam_valve_pid_sp_value := steam_valve_pid_actual_value;
END_IF

IF steam_valve_pid.eMode = E_CTRL_MODE.eCTRL_MODE_ACTIVE AND (steam_valve_pid_manual_sp <= 0) THEN
	steam_valve_pid_manual_sp := steam_valve_pid_out;
END_IF
*)
simulate_process_params.tCtrlCycleTime := T#100MS;
simulate_process_params.tTaskCycleTime := T#10MS;
simulate_process_params.fKp := simulate_process_kp;
simulate_process_params.fTheta := simulate_process_dumping_ration;
simulate_process_params.tT0 := TO_TIME(simulate_process_tT0);

simulate_process(
	fIn:= steam_valve_pid_out , 
	fManValue:= , 
	eMode:= E_CTRL_MODE.eCTRL_MODE_ACTIVE, 
	bHold:= , 
//	fOut=> steam_valve_pid_actual_value , 
	eState=> , 
	eErrorId=> , 
	bError=> , 
	stParams:= simulate_process_params);
END_ACTION

ACTION A02_WarmUp:
// Theseus - P_U01.A02_WarmUp
// Rev 1.0 - October 8, 2024

CASE i2Step OF

	0:	;
		
	1:	
		sError															:= '';
		bComplete														:= FALSE;
		bRunSteamBypass													:= FALSE;
		P_U01.steam_bypass_complete										:= FALSE;
		IF NOT P_U01.warmup_complete THEN
			gsCycleStage												:= 'warm_up.initialize';							// 3
			IF NOT TRUE THEN //P_U01.boiler_outlet_pres_error THEN
				sError													:= F_Concat3(_U01, gsCycleStage, gsBoilerError);
				i2Step													:= 80;
			ELSE
				i2Step													:= i2Step + 1;
			END_IF
		ELSE
			bComplete													:= TRUE;
			i2Step														:= 90;
		END_IF
		
	2:	
		P_U01.boiler_package												:= TRUE;											// 4
		gsCycleStage													:= 'warm_up.boiler_heating';						// 5
		P_U01.drainage_on													:= TRUE;											// 6
		bAdsorptionActive												:= FALSE;											// 7
		bAdsorptionTimer												:= FALSE;
		i2Step															:= SEL(P_U01.SP_adsorb_during_warmup, 20, i2Step + 1);	// 8

	3:
		iAxStep															:= 1;												// 8.a
		i2Step															:= i2Step + 1;

	4:	
		Ax_Process_Pre_Check();																								// 8.a																			
		IF bPreCheckDone THEN
			IF sError = '' THEN																								// 8.a.i
				P_M01.rs1.repres_valves									:= P_M01.bRS01;										// 8.b
				rTime													:= _VALVE_TIME;
				i2Step													:= i2Step + 1;
			ELSE
				P_Alarms.M_Add_Alarm(CONCAT(_U01, gsCycleStage), sError, gsWarmupWillContinueWOAdsorption);					// 8.a.ii
				i2Step													:= 20;
			END_IF
		END_IF
		
	5:
		bTimer															:= TRUE;
		bPass1															:= (P_M01.bRS01 AND P_M01.rs1.repres_valves_clear) OR NOT P_M01.bRS01;
		IF bPass1 THEN
			bTimer														:= FALSE;
			i2Step														:= i2Step + 1;
		ELSIF tonTimer.Q THEN
			bTimer														:= FALSE;
			//P_M01_RS01.close_repres_valves								:= TRUE;
			//i2Step														:= 20;
			i2Step														:= i2Step + 1; 
		END_IF
		
	6:
		P_M01.rs1.open_doors											:= P_M01.bRS01;										// 8.c
		rTime															:= P_M01.SP_doorsopenclose_timedelay * _MINUTES;	// 8.c.i
		gsCycleStage													:= 'warm_up.boiler_heating_open_doors';				// 8.c.ii
		i2Step															:= i2Step + 1;

	7:
		bTimer															:= TRUE; 
		bPass1															:= (P_M01.bRS01 AND P_M01.rs1.open_doors) OR NOT P_M01.bRS01;
		IF bPass1 THEN
			bTimer														:= FALSE;
			i2Step														:= i2Step + 1;
		ELSIF tonTimer.Q THEN
			bTimer														:= FALSE;
			sRS															:= _RS01;
			P_Alarms.M_Add_Alarm(F_Concat3(_U01, sRS, gsCycleStage), gsReactorDoorOpeningError, gsWarmupWillContinueWOAdsorption);
			i2Step														:= 20;
		END_IF

	8:
		P_M01.rs1.fan_setpoint											:= SEL(P_M01.bRS01, 0, P_M01.SP_reactor_set_1_vfd_percent);	// 8.d
		gsCycleStage													:= 'warm_up.boiler_heating_turn_on_fans';			// 8.d.i
		rTime															:= _FAN_RS_DELAY_TIME;
		i2Step															:= i2Step + 1;

	9:
		bTimer															:= TRUE;
		IF tonTimer.Q THEN
			bTimer														:= FALSE;
			i2Step														:= i2Step + 1;
		END_IF

	10:
		P_M01.rs1.r1.inlet_co2_sol										:= P_M01.bRS01;										// 8.e
		P_M01.rs1.r1.outlet_co2_sol										:= P_M01.bRS01;										// 8.e
		gsCycleStage													:= 'warm_up.boiler_heating_adsorption';				// 8.e.i
		bAdsorptionTimer												:= TRUE;											// 8.f
		bAdsorptionActive												:= TRUE;											// 8.g
		i2Step															:= 20;


//**** Complete Warmup		
	20:
		P_U01.vacuum_pres_control_valve									:= _OPEN;											// 9
		rTime															:= _VALVE_TIME;
		i2Step															:= i2Step + 1;
		
	21:	
		bTimer															:= TRUE;
		IF P_U01.vacuum_pres_control_valve_open THEN																			// 9
			bTimer														:= FALSE;
			rTime														:= P_U01.SP_boiler_warmup_duration * _MINUTES;		// 11
			i2Step														:= i2Step + 1;
		ELSIF tonTimer.Q THEN
			bTimer														:= FALSE;
			sError														:= gsProductVacuumBackfeedValveError;				// 9
			IF bAdsorptionActive THEN
				P_Alarms.M_Add_Alarm(CONCAT(_U01, gsCycleStage), sError, gsProcessCannotRunAdsorptionWillContinue);
				P_U01.boiler_package										:= FALSE;
				i2Step													:= 30;
			ELSE
				i2Step													:= 80;
			END_IF
		END_IF
		
	22:
		bTimer															:= TRUE;
		IF P_U01.boiler_ready THEN																							// 12 (Handled in P_U01.A_Points)
			bTimer														:= FALSE;
			bComplete													:= TRUE;
			P_U01.warmup_complete											:= TRUE;
			i2Step														:= i2Step + 1;
		ELSIF tonTimer.Q THEN																								// 12.a
			bTimer														:= FALSE;
			sError														:= gsBoilerError;
			i2Step														:= 80;
		END_IF

